(* CoDeSys 2.3.9.50 project: Acp_Bag_2Wrapping_Code.pro *)
(* Libraries: SysLibAlarmTrend.lib 17.10.05 13:12:38, TcBase.lib 14.5.09 12:14:08, TcSystem.lib 7.6.16 11:01:22, TcUtilities.lib 3.2.16 16:08:58, FB_DateTime.lib 15.2.16 16:36:26, STANDARD.LIB 5.6.98 12:03:02, TcEtherCAT.lib 30.11.16 19:52:18, COMlibV2.lib 24.2.14 12:45:46, SysLibTargetVisu.lib 16.6.08 16:24:26, TcBaseMath.lib 27.7.04 12:07:56, SysLibVisu.lib 7.7.04 18:17:22, TcSystemCX.lib 7.9.16 12:51:26, TcMath.lib 23.9.04 15:15:30 *)

(* Task configuration *)
TASK Standard (PRIORITY := 0, INTERVAL := T#10ms);
	MAIN
END_TASK

(* Global variable list: Alarms *)
VAR_GLOBAL
	bAError1: BOOL;
	bAError2: BOOL;
	bAError3: BOOL;
	bAError4: BOOL;
	bAError5: BOOL;
	bAError6: BOOL;
	bAError7: BOOL;
	bAError8: BOOL;
	bAError9: BOOL;
	bAError10: BOOL;
	bAError11: BOOL;
	bAError12: BOOL;
	bAError13: BOOL;
	bAError14: BOOL;
	bAError15: BOOL;
	bAError16: BOOL;
	bAError17: BOOL;
	bAError18: BOOL;
	bAError19: BOOL;
	bAError20: BOOL;
	bAError1Status: STRING;
	bAError2Status: STRING;
	bAError3Status: STRING;
	bAError4Status: STRING;
	bAError5Status: STRING;
	bAError6Status: STRING;
	bAError7Status: STRING;
	bAError8Status: STRING;
	bAError9Status: STRING;
	bAError10Status: STRING;
	bAError11Status: STRING;
	bAError12Status: STRING;
	bAError13Status: STRING;
	bAError14Status: STRING;
	bAError15Status: STRING;
	bAError16Status: STRING;
	bAError17Status: STRING;
	bAError18Status: STRING;
	bAError19Status: STRING;
	bAError20Status: STRING;
END_VAR

(* Global variable list: Auto *)
VAR_GLOBAL
	bQAFeedingConveyorMotor: BOOL;
	bAConeFeedConveyorStart: BOOL;
	bAConeFeedConWait: BOOL;
	bRConePresentInConeFeedCon: BOOL;

	bAConeFeedingPistonHomeRsError: BOOL;
	bQAConeFeedPisOn: BOOL;

	bASealConRdy: BOOL;
	bQAForwardPistonOn: BOOL;
	bQAReversePistonOn: BOOL;

	bAConeTiltingRdy: BOOL;
	ConeFeedPistonRdy: BOOL;
	bAConeFeedCount: BOOL;
	bAConeFeedPisOn: BOOL;
	bAConeFeedingPistonEndRsError: BOOL;
	Cone1Reached: BOOL;
	bAConeFeededCount: INT;
	Cone2Reached: BOOL;
	TotalNoOfCones: INT;

	bAConeFwdRevRdy: BOOL;
	bATiltingPistonOn: BOOL;
	bAConeTiltingPistonEndRsError: BOOL;
	bAFwdRevPisRdy: BOOL;
	bAFwdRevCom: BOOL;
	bAConeTiltingPistonHomeRsError: BOOL;
	bATiltingCylCom: BOOL;
	bAConeTiltingCount: INT;

	bAWrapRdy: BOOL;
	bAForwardPistonOn: BOOL;
	bAReversePistonOn: BOOL;
	bAForwardPisEndRsError: BOOL;
	bAReversePisEndRsError: BOOL;
	bAFwdRevCount: INT;
	bAForwardPisHomeRsError: BOOL;
	bAReversePisHomeRsError: BOOL;
	bAWrappingConRdy: BOOL;

	bAWrapConRdy: BOOL;
	bAWrappingConOn: BOOL;
	bAWrapConeAlaignError: BOOL;
	bAWrapConeAlaignError1: BOOL;
	bAWrappingPisRdy: BOOL;
	bAWrapPiston1On: BOOL;
	bAWrapPiston2On: BOOL;
	bASealingConRdy: BOOL;
	bASheetFeedError: BOOL;
	bAWrapPis1EndRsError: BOOL;
	bAWrapPis2EndRsError: BOOL;
	bAWrappingPisCylCom: BOOL;
	bAWrappingPisCylComInt: BOOL;
	bASealUnitStart: BOOL;


	iBagRowCounter_243: INT;
	bQAColumnStopperPiston: BOOL;
	bABagOperationStarted_243: BOOL;
	bABagUnitRdy_243: BOOL;
	bABagOperationRdy_243: BOOL;
	bQAConePusher2Piston: BOOL;
	bQAColumnReversePiston: BOOL;
	bQAConePusher1Piston: BOOL;
	bABagHalfOpCom_243: BOOL;
	bABagOperationStarted: BOOL;
	bABagOperationComplete: BOOL;
	bQABagHolder: BOOL;
	bQASeparatorplatePiston: BOOL;
	bQABagUp_Down50piston: BOOL;
	bABagOperationComplete_243: BOOL;
	bQABagPusherForwardPiston: BOOL;
	bQABagPusherReversePiston: BOOL;
	TON_bagPusher_243: TON;
	BagOpCom_243: BOOL;
	bForceBagHolder: BOOL;
	bABagComplete: BOOL;
	bQABagTiltingpistonReverse: BOOL;
	bABagTiltingRevOk_243: BOOL;
	bQAColumnConeReversePiston: BOOL;
	bQABagUp_Down180piston: BOOL;
	bQABagTiltingpistonForward: BOOL;
	bQABagBagUp_Down50piston: BOOL;
	bQABagRowHolderpiston: BOOL;

	bASealingConRdy_Bag: BOOL;
	bASealingConRdy_Box: BOOL;
	bASealingUnitOperationCom: BOOL;
	bABoxUnitRdy: BOOL;
	bABoxOperationCom: BOOL;
	bQASealingConFwd1: BOOL;
	bQASealingConRev: BOOL;
	bASealConeSet1Started: BOOL;
	bQASealingConFwd2: BOOL;
	bASealingConeCountEnable: BOOL;
	bASealConeSet1Completed: BOOL;
	bASealConeSet2Started: BOOL;
	bASealConeSet2Completed: BOOL;
	bASealConeRevSetCompleted: BOOL;
	bASealConeMissError: BOOL;
	bASealConeMissErrorStatus: STRING;
	bASealConeMissError1: BOOL;
	bASealConeMissError2: BOOL;
	bASealConeMissError3: BOOL;
	bASealingUnitInt: BOOL;
	bQASealingSeparatorYAxisPiston: BOOL;
	bQASealingTopPiston: BOOL;
	bQASealingBottomPiston: BOOL;
	bQASealingSeparatorXAxisPiston: BOOL;
END_VAR

(* Global variable list: DataLog *)
VAR_GLOBAL
	R_TRIG_IndoPrint: R_TRIG;
	FB_FileOpen_Indo: FB_FileOpen;
	FB_FileWrite_Indo: FB_FileWrite;
	FB_FileClose_Indo: FB_FileClose;
	FB_FileDelete_Indo: FB_FileDelete;
	IndoReport: INT;
	ReportHead1_Indo: BOOL;
	ST1_ProductionData: BOOL;
	ReportHead2_Indo: BOOL;
	ReportBot1_Indo: BOOL;
	stStation1_ProductionData: BOOL;
	ReportBot2_Indo: BOOL;
	testbit: BOOL;
	sOldDay: STRING;
	WriteError: INT;
	OpenError: INT;
	ProductionData_IndoPrint2:STRING(255);
	ProductionDataError_IndoPrint2:STRING(255);
	ProductionDataValues_IndoPrint_Com:STRING(255);
	bANewDay: BOOL;
	SerialNoError: DINT;
	ProductionDataValues_IndoPrint: STRING(255);
	ProductionData_IndoPrint: STRING(255);
	ProductionDataError_IndoPrint: STRING(255);
	ProductionData_ReportData1 : ProductionData_ReportData;
	PROCESSCOMPLETE: BOOL;
	ReportSave: BOOL;
	SerialNo AT %Q*: DINT;
END_VAR

(* Global variable list: Initialize *)
VAR_GLOBAL
	Initialize_TapHmi: BOOL;
	bAInitializeSeq: BOOL;
	bAMachineOn: BOOL;
	bASupplyPressureError: BOOL;
	IntAllOver: BOOL;
	bAIntHomeCheckError: BOOL;

	bQRWappingConveyorMotor: BOOL;
	WrappingConIntRunning: BOOL;
	WrapConIntOver: BOOL;
	bRConePresentInWrapCon: BOOL;
	bQRWrappingPiston1: BOOL;
	bQRWrappingPiston2: BOOL;
	bAWrappingPiston1RsError: BOOL;
	bAWrappingPiston2RsError: BOOL;
	WrapUnitIntOver: BOOL;
	sWrappingConStatus: STRING;
	TiltIntRdy: BOOL;

	bQRForwardPiston: BOOL;
	bQRReversePiston: BOOL;
	bQRTiltingPiston: BOOL;
	bQATiltingPiston: BOOL;
	TiltingIntOvr: BOOL;

	bQRSealingConveyorMotor: BOOL;
	bRConePresentInSealCon: BOOL;
	SealingConIntRunning: BOOL;
	sSealingConStatus: STRING;
	SealConIntOver: BOOL;
	bQRSealingTopPiston: BOOL;
	bQRSealingBottomPiston: BOOL;
	bQRSealingSeparatorXAxisPiston: BOOL;
	bRSealUnitIntOver: BOOL;
	bQRSealingSeparatorYAxisPiston: BOOL;

	bRBagUnitIntRdy: BOOL;
END_VAR

(* Global variable list: Inputs *)
VAR_GLOBAL
					(*I1-EL1809*)

	(*IR1*)	bIUnit_A_RowStopperHome AT %I* : BOOL;
	(*IR2*)	bIUnit_A_RowStopperMiddle AT %I* :BOOL;
	(*IR3*)	bIUnit_A_RowStopperEnd AT %I* :BOOL;
	(*IR4*)	bIUnit_B_RowStopperHome AT %I* :BOOL;
	(*IR5*)	bIUnit_B_RowStopperMiddle AT %I* :BOOL;
	(*IR6*)	bIUnit_B_RowStopperEnd AT %I* :BOOL;
	(*IR7*)	bIUnit_A_ConeDetectionSensor1 AT %I* :BOOL;
	(*IR8*)	bIUnit_A_ConeDetectionSensor2 AT %I* :BOOL;
	(*IR9*)	bIUnit_A_ConeDetectionSensor3 AT %I* :BOOL;
	(*IR10*)	bIUnit_A_ConeDetectionSensor4 AT %I* :BOOL;
	(*IR11*)	bIUnit_A_ConeCrossLimitSwitch AT %I* :BOOL;
	(*IR12*)	bIUnit_B_ConeDetectionSensor1 AT %I* :BOOL;
	(*IR13*)	bIUnit_B_ConeDetectionSensor2 AT %I* :BOOL;
	(*IR14*)	bIUnit_B_ConeDetectionSensor3 AT %I* :BOOL;
	(*IR15*)	bIUnit_B_ConeDetectionSensor4 AT %I* :BOOL;
	(*IR16*)	bIUnit_B_ConeCrossLimitSwitch AT %I* :BOOL;


					(*I2-EL1809*)

	(*IR17*)	bIUnit_AStartPb AT %I* :BOOL;
	(*IR18*)	bIUnit_BStartPb AT %I* :BOOL;
	(*IR19*)	bISpare1 AT %I* :BOOL;
	(*IW1*)	bIMcStartPb AT %I* :BOOL;
	(*IW2*)	bIMcStopPb AT %I* :BOOL;
	(*IW3*)	bIAutoManualSwitch AT %I* :BOOL;
	(*IW4*)	bIEmergencySwitchPb AT %I* :BOOL;
	(*IW5*)	bIProgramKeySwitch AT %I* :BOOL;
	(*IW6*)	bIConeOrientationTopLimitSwitch AT %I* :BOOL;
	(*IW7*)	bIFeedconeStopSensor AT %I* :BOOL;
	(*IW8*)	bIConeFeedingPistonHome AT%I* :BOOL;
	(*IW9*)	bIConeFeedingPistonEnd AT %I* :BOOL;
	(*IW10*)	bIForwardPistonHome AT %I* :BOOL;
	(*IW11*)	bIForwardPistonEnd AT %I* :BOOL;
	(*IW12*)	bIReversePistonHome AT %I* :BOOL;
	(*IW13*)	bIReversePistonEnd AT %I* :BOOL;

						(*I3-EL1809*)

	(*IW14*)	bITiltingHome AT %I* :BOOL;
	(*IW15*)	bITiltingMiddle AT %I* :BOOL;
	(*IW16*)	bITiltingEnd AT %I* :BOOL;
	(*IW17*)	bIWrappingChanelPiston1Home AT %I* :BOOL;
	(*IW18*)	bIWrappingChanelPiston1Middle AT %I* :BOOL;
	(*IW19*)	bIWrappingChanelPiston1End AT %I* :BOOL;
	(*IW20*)	bIWrappingChanelPiston2Home AT %I* :BOOL;
	(*IW21*)	bIWrappingChanelPiston2Middle AT %I* :BOOL;
	(*IW22*)	bIWrappingChanelPiston2End AT %I* :BOOL;
	(*IW23*)	bIWrappingCone1 AT %I* :BOOL;
	(*IW24*)	bIWrappingCone2 AT %I* :BOOL;
	(*IW25*)	bIFilmTensionRod1Home AT %I* :BOOL;
	(*IW26*)	bIFilmTensionRod1End AT %I* :BOOL;
	(*IW27*)	bIFilmTensionRod2Home AT %I* :BOOL;
	(*IW28*)	bIFilmTensionRod2End AT %I* :BOOL;
	(*IW29*)	bISpare2 AT %I* :BOOL;

						(*I4-EL1809*)

	(*IW30*)	bISealingSeparatorYAxisPistonHome AT %I* :BOOL;
	(*IW31*)	bISealingSeparatorYAxisPistoEnd AT %I* :BOOL;
	(*IW32*)	bISealingTopPistonHome AT %I* :BOOL;
	(*IW33*)	bISealingTopPistonEnd AT %I* :BOOL;
	(*IW34*)	bISealingBottomPistonHome AT %I* :BOOL;
	(*IW35*)	bISealingBottomPistonEnd AT %I* :BOOL;
	(*IW36*)	bISealingSeparatorXAxisPistonHome AT %I* :BOOL;
	(*IW37*)	bISealingSeparatorXAxisPistonEnd AT %I* :BOOL;
	(*IW38*)	bIManualSealingPb AT %I* :BOOL;
	(*IW39*)	bIConeCountsensor AT %I* :BOOL;
	(*IW40*)	bIPressureSwitch AT %I* :BOOL;
	(*IW41*)	bIResetPb AT %I* :BOOL;
	(*IW42*)	bIPausePb AT %I* :BOOL;
	(*IW43*)	bIConeCountSensorRev AT %I* :BOOL;
	(*IW44*)	bIConecountStopperPistonHome AT %I* :BOOL;
	(*IW45*)	bIConecountStopperPistonEnd AT%I* :BOOL;


						(*I5-EL1809*)

	(*IW46*)	bIResetSealingPb AT %I* :BOOL;
	(*IW47*)	bISpare4 AT %I* :BOOL;
	(*IW48*)	bISpare5 AT %I* :BOOL;
	(*IW49*)	bISpare6 AT %I* :BOOL;
	(*IW50*)	bISpare7 AT %I* :BOOL;
	(*IW51*)	bISpare8 AT %I* :BOOL;
	(*IW52*)	bISpare9 AT %I* :BOOL;
	(*IW53*)	bISpare10 AT %I*: BOOL;

					(*I6-EL1809*)

	(*IB1*)	bIColumnStopperPistonHome AT %I*: BOOL;
	(*IB2*)	bIColumnStopperPistonEnd AT %I*: BOOL;
	(*IB3*)	bIColumnReversePistonHome AT %I*: BOOL;
	(*IB4*)	bIColumnReversePistonEnd AT %I*: BOOL;
	(*IB5*)	bISeperatorPlatePistonHome AT %I*: BOOL;
	(*IB6*)	bISeperatorPlatePistonEnd AT %I*: BOOL;
	(*IB7*)	bIConePusher1PistonHome AT %I*: BOOL;
	(*IB8*)	bIConePusher1PistonEnd AT %I*: BOOL;
	(*IB9*)	bIConePusher1SaftyObjectSensor AT %I*: BOOL;
	(*IB10*)	bIBagUpDown180PistonHome AT %I*: BOOL;
	(*IB11*)	bIBagUpDown180PistonEnd AT %I*: BOOL;
	(*IB12*)	bIBagUpDown50PistonHome AT %I*: BOOL;
	(*IB13*)	bIBagUpDown50PistonEnd AT %I*: BOOL;
	(*IB14*)	bIBagPusherPistonHome AT %I*: BOOL;
	(*IB15*)	bIBagPusherPistonMiddle AT %I*: BOOL;
	(*IB16*)	bIBagPusherPistonEnd AT %I*: BOOL;

						(*I7-EL1809*)

	(*IB17*)	bIBagTiltingPistonHome AT %I*: BOOL;
	(*IB18*)	bIBagiltingPistonEnd AT %I*: BOOL;
	(*IB19*)	bIBagEmptyCheckObjectSensor AT %I*: BOOL;
	(*IB20*)	bIBagHolderOn  AT %I*: BOOL;
	(*IB21*)	bIBagResetPb AT %I*: BOOL;
	(*IB22*) 	bISpare11 AT %I*: BOOL;
	(*IB23*) 	bISpare12 AT %I*: BOOL;
	(*IB24*) 	bISpare13 AT %I*: BOOL;
END_VAR

(* Global variable list: Main *)
VAR_GLOBAL
	(****************START / STOP / PAUSE / RESUME***************)
	Start_TapHmi: BOOL;
	bAutoModeOn: BOOL;
	bMcStartInAuto: BOOL;
	bMcStopEnable: BOOL;
	Stop_TapHmi: BOOL;
	Pause_TapHmi: BOOL;
	bPauseSeq: BOOL;
	Resume_TapHmi: BOOL;
	Reset_TapHmi: BOOL;
	bErrorReset: BOOL;
	bMcStopEnable1: BOOL;
(*============== Auto/Manual Mode Selection Logic========================*)
	bManualModeOn: BOOL;
	bManualmode: BOOL;
	sMcStatus: STRING;
	bHidePopUp: BOOL;
	bManualModeOk_TapHmi: BOOL;
	bManualModeNOk_TapHmi: BOOL;
(*====================Logic for Model Selection===============*)
	BagSelect_TapHmi: BOOL;
	bAMainIntStarted: BOOL;
	bABoxModeSelected: BOOL;
	BoxSelect_TapHmi: BOOL;
	bABagModeSelected: BOOL;
	sPackingModeStatus: STRING;

	(****************DATE AND TIME***********)
	FB_DateTime_1: FB_DateTime;
	sHourPreFix: STRING;
	sHou: STRING;
	sDayPreFix: STRING;
	sDay: STRING;
	sMonthPreFix: STRING;
	sMonth: STRING;
	sDayF: STRING;
	sMonthF: STRING;
	sDayMonth: STRING;
	sDayF1: STRING;
	sMonthF1: STRING;
	sDayMonth1: STRING;
	sDayMonthYear: STRING;
	sDayMonthYear1: STRING;
	sDaateReport: STRING;
	ReportPath: STRING;
	ReportPath_Final: STRING;
	ReportPath_Final_1: STRING;
	ReportPath_Final_2: STRING;
	sDateReport: STRING;
	ReportPathError: STRING;
	ReportPath_FinalError: STRING;
	ReportPath_Final_1Error: STRING;
	ReportPath_Final_2Error: STRING;
	DateTimeVar: STRING;
	wTodayToHmiFinal: STRING;
(*===============Shift Calculation============*)
	bAShift1Hour: BOOL;
	bAShift2Hour: BOOL;
	bAShift3Hour: BOOL;
	Sfiht1From_Hmi  AT %Q*: WORD;
	Sfiht2From_Hmi  AT %Q*: WORD;
	Sfiht3From_Hmi  AT %Q*: WORD;
	Sfiht1To_Hmi AT %Q*: WORD;
	Sfiht2To_Hmi AT %Q*: WORD;
	Sfiht3To_Hmi AT %Q*: WORD;
	sShitStatus: STRING;
END_VAR

(* Global variable list: Manual *)
VAR_GLOBAL
	WrappingSafety: BOOL;
	SealingSafety: BOOL;
	bManualSealEnable: BOOL;
	bManualSealEnable2: BOOL;
	bMManualSealOn: BOOL;
	bQM_Cone_Sealing_Bottom_Piston: BOOL;
	bQM_Cone_Sealing_Top_Piston: BOOL;
	bHMI_Cone_Forward_Piston_On: BOOL;
	bQM_Cone_Forward_Piston: BOOL;
	bHMI_Cone_Feeding_Piston_On: BOOL;
	bQM_Cone_Feeding_Piston: BOOL;
	bHMI_Cone_Reverse_Piston_On: BOOL;
	bQM_Cone_Reverse_Piston: BOOL;
	bHMI_Cone_Tilting_Piston_On: BOOL;
	bQM_Cone_Tilting_Piston: BOOL;
	bQM_Cone_Tilting_Piston_Rev: BOOL;
	bHMI_Cone_Tilting_Piston_On_Rev: BOOL;
	bHMI_Cone_Wrapping_Piston_On: BOOL;
	bQM_Cone_Wrapping_Piston_Rev: BOOL;
	bQM_Cone_Wrapping_Piston_Fwd: BOOL;
	bHMI_Cone_Wrapping_Piston_On_Rev: BOOL;
	bHMI_Cone_Sealing_Top_Piston_On: BOOL;
	bHMI_Cone_Sealing_Bottom_Piston_On: BOOL;
	bHMI_Cone_Sealing_YAxis_Piston_On: BOOL;
	bQM_Cone_Sealing_YAxis_Piston: BOOL;
	bHMI_Cone_Sealing_XAxis_Piston_On: BOOL;
	bQM_Cone_Sealing_XAxis_Piston: BOOL;
	bHMI_Cone_Feeding_Conveyor_On: BOOL;
	bQM_Cone_Feeding_Conveyor: BOOL;
	bHMI_Cone_Wrapping_Conveyor_On: BOOL;
	bQM_Cone_Wrapping_Conveyor: BOOL;
	bHMI_Cone_Sealing_Conveyor_On: BOOL;
	bQM_Cone_Sealing_Conveyor: BOOL;
	bIConePusher1_On_Hmi: BOOL;
	bQMConePusher1: BOOL;
	bIConePusher2_On_Hmi: BOOL;
	bQMConePusher2: BOOL;
	bIConePusher3_On_Hmi: BOOL;
	bQMConePusher3: BOOL;
	bIBagPusherFwd_On_Hmi: BOOL;
	bQMBagPusherFwd: BOOL;
	bIBagPusherRev_On_Hmi: BOOL;
	bQMBagPusherRev: BOOL;
	bIUpDownPiston_1_On_Hmi: BOOL;
	bQMUpDownPiston_1: BOOL;
	bIUpDownPiston_2_On_Hmi: BOOL;
	bQMUpDownPiston_2: BOOL;
	bIBagTiltingFwd_On_Hmi: BOOL;
	bQMBagTiltingFwd: BOOL;
	bIBagTiltingRev_On_Hmi: BOOL;
	bQMBagTiltingRev: BOOL;
	bIColumn_Stopper_Piston_On_Hmi: BOOL;
	bQMColumnStopperPiston: BOOL;
	bIColumnConeForwardPiston_On_Hmi: BOOL;
	bQMColumnConeForwardPiston: BOOL;
	bIBagHolder_On: BOOL;
	bIBagHolder_On_Hmi: BOOL;
	bIBagPusherHome: BOOL;
	bQMBagHolderPiston: BOOL;
	bHMI_RetA_Fwd_On: BOOL;
	bHMI_RetA_Rev_On: BOOL;
	bQM_RetA_Rev: BOOL;
	bQM_RetA_Fwd: BOOL;
	bHMI_Ret_RevA_On: BOOL;

	bHMI_RetB_Fwd_On: BOOL;
	bHMI_RetB_Rev_On: BOOL;
	bQM_RetB_Rev: BOOL;
	bQM_RetB_Fwd: BOOL;
	bHMI_Ret_RevB_On: BOOL;
	bHMI_Cone_Wrapping_Piston1_On: BOOL;
	bQM_Cone_Wrapping_Piston1_Fwd: BOOL;
	bHMI_Cone_Wrapping_Piston1_On_Rev: BOOL;
	bQM_Cone_Wrapping_Piston1_Rev: BOOL;
	bHMI_Cone_Wrapping_Piston2_On: BOOL;
	bQM_Cone_Wrapping_Piston2_Rev: BOOL;
	bQM_Cone_Wrapping_Piston2_Fwd: BOOL;
	bHMI_Cone_Wrapping_Piston2_On_Rev: BOOL;
END_VAR

(* Global variable list: Outputs *)
VAR_GLOBAL
				(*O1-EL2809*)

	RetA_RowStopperMotorFwd AT %Q* :BOOL;(*OR1*)
	RetA_RowStopperMotorRev AT %Q* :BOOL;(*OR2*)
	RetB_RowStopperMotorFwd AT %Q* :BOOL;(*OR3*)
	RetB_RowStopperMotorRev AT %Q* :BOOL;(*OR4*)
	SpareOutput1 AT %Q* :BOOL;(*OR5*)
	RetA_WeightOk AT %Q* :BOOL;(*OR6*)
	RetA_WeightNOk AT %Q* :BOOL;(*OR7*)
	RetB_WeightOk AT %Q* :BOOL;(*OR8*)
	RetB_WeightNOk AT %Q* :BOOL;(*OR9*)
	SpareOutput2 AT %Q* :BOOL;(*OR10*)
	SpareOutput3 AT %Q* :BOOL;(*OR11*)
	SpareOutput4 AT %Q* :BOOL;(*OR12*)
	TowerLampRed AT %Q* :BOOL;(*R1*)
	TowerLampGreen AT %Q* :BOOL;(*R2*)
	TowerLampYellow AT %Q* :BOOL;(*R3*)
	TowerBuzzer AT %Q* :BOOL;(*R4*)


			(*O2-EL2809*)

	ConeFeedingPiston AT %Q* :BOOL;(*OW1*)
	ForwardPiston AT %Q* :BOOL;(*OW2*)
	ReversePiston AT %Q* :BOOL;(*OW3*)
	TiltingPiston AT %Q* :BOOL;(*OW4*)
	WrappingPiston1 AT %Q* :BOOL;(*OW5*)
	WrappingPiston2 AT %Q* :BOOL;(*OW6*)
	SealingSeparatorYAxisPiston AT %Q* :BOOL;(*OW7*)
	SealingTopPiston AT %Q* :BOOL;(*OW8*)
	SealingBottomPiston AT %Q* :BOOL;(*OW9*)
	SealingSeparatorXAxisPiston AT %Q* :BOOL;(*OW10*)
	FilmRollerMotor1 AT %Q* :BOOL;(*OW11*)
	FilmRollerMotor2 AT %Q* :BOOL;(*OW12*)
	ConeCountPiston AT %Q* :BOOL;(*OW13*)
	FeedingConveyorMotor AT %Q* :BOOL;(*OW14*)
	WappingConveyorMotor AT %Q* :BOOL;(*OW15*)
	SealingConveyorMotor AT %Q* :BOOL;(*OW16*)



			(*O3-EL2008*)

	SpareOutput5 AT %Q* :BOOL;(*OW20*)
	SpareOutput6 AT %Q* :BOOL;(*OW21*)
	SpareOutput7 AT %Q* :BOOL;(*OW22*)
	SpareOutput8 AT %Q* :BOOL;(*OW23*)
	SpareOutput9 AT %Q* :BOOL;(*OW24*)
	SpareOutput10 AT %Q* :BOOL;(*OW25*)
	SpareOutput11 AT %Q* :BOOL;(*OW26*)
	SpareOutput12 AT %Q* :BOOL;(*OW27*)

			(*O4-EL2809*)

	ColumnStopperPiston AT %Q* :BOOL;(*OB1*)
	ColumnReversePiston AT %Q* :BOOL;(*OB2*)
	SeparatorplatePiston AT %Q* :BOOL;(*OB3*)
	ConePusher1Piston AT %Q* :BOOL;(*OB4*)
	ConePusher2Piston AT %Q* :BOOL;(*OB5*)
	BagPusherForwardPiston AT %Q* :BOOL;(*OB6*)
	BagPusherReversePiston AT %Q* :BOOL;(*OB7*)
	BagHolderpiston AT %Q* :BOOL;(*OB8*)
	BagUp_Down180piston AT %Q* :BOOL;(*OB9*)
	BagUp_Down50piston AT %Q* :BOOL;(*OB10*)
	BagTiltingpistonForward AT %Q* :BOOL;(*OB11*)
	BagTiltingpistonReverse AT %Q* :BOOL;(*OB12*)
	BagRowHolderpiston AT %Q* :BOOL;(*OB13*)
	SpareOutput13 AT %Q* :BOOL;(*OB14*)
	SpareOutput14 AT %Q* :BOOL;(*OB15*)
	SpareOutput15 AT %Q* :BOOL;(*OB16*)

END_VAR

(* Global variable list: Parameters *)
VAR_GLOBAL
	Default_NetWeight_Report: STRING;
	Default_GrossWeight_Report: STRING;
	Actual_NetWeight_Report: STRING;
	Actual_GrossWeight_Report: STRING;
	COUNT_DIS: STRING;
	BLEND_DIS: STRING;
	LOTNO_DIS: STRING;
	CARTONNO_DIS: DINT;
	SHADE_DIS: STRING;
END_VAR

(* Global variable list: Print *)
VAR_GLOBAL
	PrintEnabled: BOOL;
	PrintValue: INT;
	PrintEnable_TogHmi: BOOL;
	ProductionData_PrintData: ProductionData_PrintData;
	ProductionDataValues_Print: STRING(255);
	ProductionDataValues_Print_Com:STRING(255);
	ProductionData_Print: STRING(255);
	FB_FileOpen1: FB_FileOpen;
	FB_FileWrite1: FB_FileWrite;
	FB_FileClose1: FB_FileClose;
	FB_FileDelete1: FB_FileDelete;
	PrintOk: BOOL;
END_VAR

(* Data type *)
TYPE ProductionData_PrintData :
STRUCT
	Print:STRING;
	ConeType1:STRING;
	Blend1:STRING;
	DefaultnetWt1:STRING;
	DefaultGrossWt1:STRING;
	LotNo1:STRING;
	BagNo1:STRING;
	Shade1:STRING;
END_STRUCT
END_TYPE

(* Data type *)
TYPE ProductionData_ReportData :
STRUCT
	SERIALNO			:STRING;
	SDATE				:STRING;
	STIME				:STRING;
	BAGNO				:STRING;
	COUNTCODE		:STRING;
	LOTNO				:STRING;
	DFLTNETWEIGHT	:STRING;
	ACTNETWEIGHT		:STRING;
	DFLTGROSSWEIGHT	:STRING;
	ACTGROSSWEIGHT	:STRING;
END_STRUCT
END_TYPE

(* POU MAIN, ST *)
PROGRAM MAIN
	VAR

END_VAR
					(*START / STOP / PAUSE / RESUME*)


	IF (bIMcStartPb OR Start_TapHmi)  AND bAutoModeOn  THEN
	 bMcStartInAuto:=TRUE;
	bMcStopEnable:=FALSE;
	END_IF

	IF  bIMcStopPb OR Stop_TapHmi  OR NOT bAutoModeOn OR NOT bIEmergencySwitchPb THEN
	 bMcStartInAuto:=FALSE;bMcStopEnable:=TRUE;bMcStopEnable1:=TRUE;
	ELSE bMcStopEnable1:=TRUE;
	 END_IF

	IF Pause_TapHmi THEN
	bPauseSeq:=TRUE;END_IF
	IF Resume_TapHmi THEN
	bPauseSeq:=FALSE;END_IF

	IF bIResetPb OR Reset_TapHmi  OR bIResetSealingPb THEN
	bErrorReset:=TRUE;
	ELSE bErrorReset:=FALSE;END_IF

					(*============== Auto/Manual Mode Selection Logic========================*)

		IF bIAutoManualSwitch THEN
			bAutoModeOn:=TRUE; bManualModeOn:=FALSE;
		ELSIF  bManualmode  THEN
			bManualModeOn:=TRUE; bAutoModeOn:=FALSE;
		END_IF

		IF bManualModeOn THEN sMcStatus:='Machine in Manual Mode';
		ELSIF bAutoModeOn THEN sMcStatus:='Machine in Auto Mode';
		END_IF

	IF bMcStartInAuto  AND NOT  bIAutoManualSwitch THEN
	bHidePopUp:=TRUE; END_IF

	IF NOT  bMcStartInAuto  AND NOT  bIAutoManualSwitch THEN
	bManualmode:=TRUE;  END_IF

	IF bHidePopUp AND bManualModeOk_TapHmi THEN
	bManualmode:=TRUE;bAutoModeOn:=FALSE;bHidePopUp:=FALSE; END_IF

	IF bHidePopUp AND bManualModeNOk_TapHmi THEN
	bHidePopUp:=FALSE; END_IF

					 (*====================Logic for Model Selection===============*)

		IF bAutoModeOn AND BagSelect_TapHmi AND NOT bAMainIntStarted THEN
		bABoxModeSelected:=FALSE;BoxSelect_TapHmi:=FALSE;bABagModeSelected:=TRUE; BoxSelect_TapHmi:=FALSE;
		ELSIF bAutoModeOn AND   BoxSelect_TapHmi AND NOT bAMainIntStarted THEN
		bABagModeSelected:=FALSE; BagSelect_TapHmi:=FALSE;bABoxModeSelected:=TRUE;
		END_IF

		IF bABagModeSelected THEN sPackingModeStatus:=' Bag Packing Selected '; END_IF
		IF bABoxModeSelected THEN sPackingModeStatus:=' Carton Packing Selected  '; END_IF




			(****************DATE AND TIME***********)

(*======================= RTC==============================*)

FB_DateTime_1(NET_ID:='5.62.177.154.1.1 ' , DATE_TIME=> );

IF FB_DateTime_1.FBLTIME.systemTime.wHour >0 AND  FB_DateTime_1.FBLTIME.systemTime.wHour<9 THEN
sHourPreFix:='0';sHou:=CONCAT(STR1:=sHourPreFix, Str2:=WORD_TO_STRING(FB_DateTime_1.FBLTIME.systemTime.wHour));
ELSIF FB_DateTime_1.FBLTIME.systemTime.wHour >=10 AND  FB_DateTime_1.FBLTIME.systemTime.wHour<=24 THEN
sHou:=WORD_TO_STRING(FB_DateTime_1.FBLTIME.systemTime.wHour);
END_IF

IF FB_DateTime_1.FBLTIME.systemTime.wDay >0 AND  FB_DateTime_1.FBLTIME.systemTime.wDay<10 THEN
sDayPreFix:='0';sDay:=CONCAT(STR1:=sDayPreFix, Str2:=WORD_TO_STRING(FB_DateTime_1.FBLTIME.systemTime.wDay));
ELSIF FB_DateTime_1.FBLTIME.systemTime.wDay >=10 AND  FB_DateTime_1.FBLTIME.systemTime.wDay<=31 THEN
sDay:=WORD_TO_STRING(FB_DateTime_1.FBLTIME.systemTime.wDay);
END_IF

IF FB_DateTime_1.FBLTIME.systemTime.wMonth >0 AND  FB_DateTime_1.FBLTIME.systemTime.wMonth<10 THEN
sMonthPreFix:='0';sMonth:=CONCAT(STR1:=sMonthPreFix, Str2:=WORD_TO_STRING(FB_DateTime_1.FBLTIME.systemTime.wMonth));
ELSIF FB_DateTime_1.FBLTIME.systemTime.wMonth >=10 AND  FB_DateTime_1.FBLTIME.systemTime.wMonth<=12 THEN
sMonth:=WORD_TO_STRING(FB_DateTime_1.FBLTIME.systemTime.wMonth);
END_IF

sDayF1:=CONCAT(STR1:=sDay, STR2:=':');
sMonthF1:=CONCAT(STR1:=sMonth, STR2:=':');
sDayMonth1:=CONCAT(STR1:=sDayF1, STR2:=sMonthF1);
sDayMonthYear1:=CONCAT(STR1:=sDayMonth1, STR2:=WORD_TO_STRING(FB_DateTime_1.FBLTIME.systemTime.wYear));

sDaateReport:=(sDayMonthYear1);

sDayF:=CONCAT(STR1:=sDay, STR2:='_');
sMonthF:=CONCAT(STR1:=sMonth, STR2:='_');
sDayMonth:=CONCAT(STR1:=sDayF, STR2:=sMonthF);
sDayMonthYear:=CONCAT(STR1:=sDayMonth, STR2:=WORD_TO_STRING(FB_DateTime_1.FBLTIME.systemTime.wYear));

ReportPath:=CONCAT(STR1:='ProductionData', STR2:='_');
ReportPath_Final:=CONCAT(STR1:=ReportPath, STR2:=sDayMonthYear);

ReportPath_Final_1:=CONCAT(STR1:='\\computer-PC\Reports\', STR2:=ReportPath_Final);
ReportPath_Final_2:=CONCAT(STR1:=ReportPath_Final_1, STR2:='.csv');

sDayF1:=CONCAT(STR1:=sDay, STR2:=':');
sMonthF1:=CONCAT(STR1:=sMonth, STR2:=':');
sDayMonth1:=CONCAT(STR1:=sDayF1, STR2:=sMonthF1);
sDayMonthYear1:=CONCAT(STR1:=sDayMonth1, STR2:=WORD_TO_STRING(FB_DateTime_1.FBLTIME.systemTime.wYear));

sDateReport:=(sDayMonthYear1);

sDayF:=CONCAT(STR1:=sDay, STR2:='_');
sMonthF:=CONCAT(STR1:=sMonth, STR2:='_');
sDayMonth:=CONCAT(STR1:=sDayF, STR2:=sMonthF);
sDayMonthYear:=CONCAT(STR1:=sDayMonth, STR2:=WORD_TO_STRING(FB_DateTime_1.FBLTIME.systemTime.wYear));

ReportPathError:=CONCAT(STR1:='ErrorData', STR2:='_');
ReportPath_FinalError:=CONCAT(STR1:=ReportPathError, STR2:=sDayMonthYear);

ReportPath_Final_1Error:=CONCAT(STR1:='\\computer-PC\Reports\', STR2:=ReportPath_FinalError);
ReportPath_Final_2Error:=CONCAT(STR1:=ReportPath_Final_1Error, STR2:='.csv');

DateTimeVar:=FB_DateTime_1.DATE_TIME;



					(*===============Shift Calculation============*)


IF FB_DateTime_1.FBLTIME.systemTime.wHour >= Sfiht1From_Hmi AND FB_DateTime_1.FBLTIME.systemTime.wHour<=Sfiht1To_Hmi THEN
bAShift1Hour:=TRUE;
ELSE
bAShift1Hour:=FALSE;
END_IF



IF FB_DateTime_1.FBLTIME.systemTime.wHour>=Sfiht2From_Hmi AND FB_DateTime_1.FBLTIME.systemTime.wHour <= Sfiht2To_Hmi THEN

bAShift2Hour:=TRUE;
ELSE
bAShift2Hour:=FALSE;
END_IF


IF FB_DateTime_1.FBLTIME.systemTime.wHour>=  Sfiht3From_Hmi AND FB_DateTime_1.FBLTIME.systemTime.wHour<=  Sfiht3To_Hmi THEN

bAShift3Hour:=TRUE;
ELSE
bAShift3Hour:=FALSE;
END_IF

IF bAShift1Hour THEN sShitStatus:='SHIFT - 1';
ELSIF bAShift2Hour THEN sShitStatus:='SHIFT - 2';
ELSIF bAShift3Hour THEN sShitStatus:='SHIFT - 3';
END_IF

Bag_Unit();
ConeFeedCon();
ConeFeedPiston();
Forward_Reverse_Piston();
Ret_A();
Ret_B();
Sealing_Unit();
Tilting_Piston();
Wrapping_Unit();
ErrorData_Report();
Print_Report();
ProductionData_Report();
Bag_Int();
ConeFeedCon_Int();
ConeTransfer_Int();
Main_Int();
Ret_Int();
Sealing_Int();
Wrapping_Int();
Manual();
Weight_Read();
END_PROGRAM

(* POU Auto/Bag_Unit, ST *)
PROGRAM Bag_Unit
VAR
	step: INT;
	iBagRowCounter_243: INT;
	TON_ConeFeedFwdOffDly_1_243: TON;
	TON_Count_243: TON;
	TON_ConePusherOffDly_243: TON;
	TON_ConeFeedFwdOffDly_243: TON;
	TON_ConePusherOnDly_243: TON;
	TON_ConePusherOffDly_2_243: TON;
	TON_ConeFeedFwdOffDly_3_243: TON;
	TON_ConePusherOnDly_2_243: TON;
	TON_ConePusherOnDly_3_243: TON;
	TON_bagPusher_243: TON;
	BagTilting_Blink2_243: TON;
	BagTilting_Blink1_243: TON;

END_VAR
CASE step OF

0:IF IntAllOver AND bABagModeSelected THEN iBagRowCounter_243:= 0; step:=step+1;END_IF

1:	iBagRowCounter_243:= 0; step:=step+1;

2:	bQAColumnConeReversePiston:=FALSE;
	IF bIColumnReversePistonHome AND NOT bPauseSeq THEN
	TON_ConeFeedFwdOffDly_1_243(IN:=FALSE); step := step +1;END_IF

3:	TON_ConeFeedFwdOffDly_1_243(IN:=TRUE , PT:=t#0.1s , Q=> , ET=> );
	IF  TON_ConeFeedFwdOffDly_1_243.Q THEN step := step +1;END_IF

4:	TON_ConeFeedFwdOffDly_1_243(IN:=FALSE);bQAColumnStopperPiston:=TRUE;
	IF  bIColumnStopperPistonEnd AND NOT bPauseSeq THEN
		 bABagOperationStarted_243:= FALSE;bABagUnitRdy_243:=TRUE;
		step := step +1;
	END_IF

5:	IF bABagOperationRdy_243  AND NOT bPauseSeq THEN
	 iBagRowCounter_243:=iBagRowCounter_243+1;bABagOperationStarted_243:=TRUE;
	bABagOperationRdy_243:=FALSE; step:=step+1;
	END_IF

6:	TON_Count_243(IN:=FALSE);bABagOperationRdy_243:=FALSE;
	IF (iBagRowCounter_243 = 1 OR iBagRowCounter_243= 2 OR iBagRowCounter_243 = 3 OR iBagRowCounter_243 = 4 ) AND NOT bPauseSeq THEN
	step:=step+1;

	ELSIF  ( iBagRowCounter_243 = 5 OR  iBagRowCounter_243 = 6 OR  iBagRowCounter_243 = 7 OR iBagRowCounter_243 = 8 ) AND NOT bPauseSeq THEN
	step := 19;
	END_IF

7:	IF   bISeperatorPlatePistonHome AND bIConePusher1PistonHome AND bIBagPusherPistonHome AND bIBagUpDown50PistonEnd
	AND bIBagUpDown180PistonEnd AND bIColumnStopperPistonEnd AND NOT bQABagHolder  AND NOT bPauseSeq THEN
	bQAConePusher2Piston:=FALSE;
	step := step +1;
	END_IF

8:	TON_ConePusherOffDly_243(IN:=TRUE , PT:=t#1s , Q=> , ET=> );
	IF TON_ConePusherOffDly_243.Q  AND NOT bPauseSeq  THEN
	bQAColumnReversePiston:=TRUE;
	TON_ConeFeedFwdOffDly_243(IN:=TRUE , PT:=t#0.1s , Q=> , ET=> );
	IF  TON_ConeFeedFwdOffDly_243.Q AND  bIColumnReversePistonEnd THEN step := step +1;END_IF
	END_IF

9:	TON_ConePusherOffDly_243(IN:=FALSE);
	IF  NOT bPauseSeq  THEN bQAColumnStopperPiston:=FALSE;step := step +1;END_IF

10:	TON_ConeFeedFwdOffDly_243(IN:=FALSE);
	IF bIColumnStopperPistonHome AND NOT bPauseSeq  THEN TON_ConePusherOnDly_243(IN:=TRUE , PT:=t#0.2s , Q=> , ET=> );
	IF TON_ConePusherOnDly_243.Q AND NOT bPauseSeq THEN
 		bQAConePusher1Piston:= TRUE ;bQAColumnReversePiston:=FALSE;step := step +1;
	END_IF END_IF

11: TON_ConePusherOnDly_243(IN:=FALSE);
	 IF bIConePusher1PistonEnd AND bIColumnReversePistonHome AND NOT bPauseSeq THEN
		bQAConePusher2Piston:= TRUE;bABagHalfOpCom_243:=TRUE;step := step +1;
	END_IF

12:	TON_ConePusherOnDly_243(IN:=TRUE , PT:=t#1.5s , Q=> , ET=> );
	IF TON_ConePusherOnDly_243.Q  AND NOT bPauseSeq  THEN bQAConePusher1Piston:= FALSE;
			step := step +1;
	END_IF

13:	TON_ConePusherOnDly_243(IN:=FALSE);
	 IF bIConePusher1PistonHome AND  (iBagRowCounter_243 = 1 OR iBagRowCounter_243 = 2  OR  iBagRowCounter_243 = 3 )
	AND NOT bQABagHolder  AND NOT bPauseSeq THEN
	bQAColumnStopperPiston:=TRUE;
		IF bIColumnStopperPistonEnd AND NOT bPauseSeq THEN
		 bABagOperationStarted:= FALSE;bABagOperationComplete:=TRUE;
		step := 2;END_IF

		ELSIF bIConePusher1PistonHome AND iBagRowCounter_243 =4  AND NOT bQABagHolder  AND NOT bPauseSeq THEN bQAColumnStopperPiston:=FALSE;
		IF  bIColumnStopperPistonHome AND NOT bPauseSeq THEN
		bABagOperationStarted_243:= FALSE;bABagOperationComplete_243:=TRUE;
		step :=14 ;END_IF
	END_IF

14:	step := step +1;

15:	IF   bISeperatorPlatePistonHome AND  bIConePusher1PistonHome AND bIBagPusherPistonHome AND NOT bPauseSeq AND NOT bQABagHolder THEN
	bQABagUp_Down180piston:=FALSE; step := step+1;bQAColumnStopperPiston:=TRUE;

	END_IF

16:	 IF bIBagUpDown180PistonHome AND bISeperatorPlatePistonHome AND bIConePusher1PistonHome AND NOT bQABagHolder  AND NOT bPauseSeq THEN
	bQASeparatorplatePiston:= TRUE ;bQABagUp_Down50piston:=FALSE;step := step +1;
	END_IF

17:	 IF bISeperatorPlatePistonEnd AND bIConePusher1PistonHome AND bIBagPusherPistonHome AND bIBagUpDown180PistonHome
	AND bIColumnStopperPistonEnd AND NOT bQABagHolder  AND NOT bPauseSeq THEN
	bQABagTiltingpistonForward:=TRUE;bQABagBagUp_Down50piston:=TRUE;bQABagTiltingpistonReverse:=FALSE;
	step := step +1;END_IF

18:	bQAColumnStopperPiston:=TRUE;
	 IF bISeperatorPlatePistonEnd AND bIConePusher1PistonHome AND bIBagPusherPistonHome AND bIBagUpDown50PistonEnd AND bIColumnStopperPistonEnd
	AND NOT bQABagHolder  AND NOT bPauseSeq THEN
	step := 2;END_IF

19:	bQAConePusher2Piston:= FALSE;step := step +1;


20:	TON_ConePusherOffDly_2_243(IN:=TRUE , PT:=t#1s , Q=> , ET=> );
	IF TON_ConePusherOffDly_2_243.Q  AND NOT bPauseSeq  THEN step := step +1;
	END_IF

21:	TON_ConePusherOffDly_2_243(IN:=FALSE);
	 IF bISeperatorPlatePistonEnd AND bIConePusher1PistonHome AND bIBagPusherPistonHome AND
	bIBagUpDown50PistonEnd AND bIColumnStopperPistonEnd AND
	bIColumnReversePistonHome AND NOT bQABagHolder  AND NOT bPauseSeq THEN
	bQAColumnReversePiston:=TRUE;step := step +1;END_IF

22:	TON_ConeFeedFwdOffDly_3_243(IN:=TRUE , PT:=t#0.1s , Q=> , ET=> );
	IF  TON_ConeFeedFwdOffDly_3_243.Q AND  bIColumnReversePistonEnd THEN step := step +1;END_IF

23:	TON_ConeFeedFwdOffDly_3_243(IN:=FALSE);bQAColumnStopperPiston:=FALSE;step := step +1;

24:	IF bIColumnStopperPistonHome AND NOT bPauseSeq  THEN TON_ConePusherOnDly_2_243(IN:=TRUE , PT:=t#0.2s , Q=> , ET=> );
	IF TON_ConePusherOnDly_2_243.Q AND NOT bPauseSeq THEN
	bQAConePusher1Piston:= TRUE ;bQAColumnReversePiston:=FALSE;step := step +1;
	END_IF END_IF
25:	TON_ConePusherOnDly_2_243(IN:=FALSE);
	 IF bIConePusher1PistonEnd AND bIColumnReversePistonHome AND NOT bQABagHolder  AND NOT bPauseSeq THEN
	bQAConePusher2Piston:= TRUE;bABagHalfOpCom_243:=TRUE;step := step +1;
	END_IF

26:	TON_ConePusherOnDly_3_243(IN:=TRUE , PT:=t#1.5s , Q=> , ET=> );
	IF TON_ConePusherOnDly_3_243.Q  AND NOT bPauseSeq  THEN
			step := step +1;
	END_IF

27:TON_ConePusherOnDly_3_243(IN:=FALSE);
	 IF bIConePusher1PistonEnd AND (iBagRowCounter_243 = 5 OR iBagRowCounter_243 = 6 OR iBagRowCounter_243 = 7  )
	AND NOT bQABagHolder  AND NOT bPauseSeq THEN
	bQAConePusher1Piston:= FALSE;step := step +1;
	ELSIF
	 bIConePusher1PistonEnd AND iBagRowCounter_243 = 8  AND NOT bQABagHolder  AND NOT bPauseSeq THEN
	step := 29;
	END_IF

28:IF  bIConePusher1PistonHome AND bIColumnStopperPistonHome THEN  bQAColumnStopperPiston:=TRUE;
	bABagOperationStarted_243:= FALSE; bABagOperationComplete_243:=TRUE;
	step := 2;END_IF

29: IF bIConePusher1PistonEnd AND bIBagUpDown50PistonEnd   AND NOT  bQABagHolder AND NOT bPauseSeq THEN
	bQABagPusherForwardPiston:=TRUE;bQABagPusherReversePiston:=FALSE;step := step +1;END_IF

30:TON_bagPusher_243(IN:=TRUE , PT:=t#0.4s , Q=> , ET=> );
	IF (TON_bagPusher_243.Q OR bIBagPusherPistonMiddle) THEN bQABagPusherForwardPiston:=FALSE;bQABagPusherReversePiston:=FALSE; step := step +1;END_IF

31:	TON_bagPusher_243(IN:=FALSE);
	bQABagPusherForwardPiston:=FALSE;bQABagPusherReversePiston:=FALSE;step := step +1;(*END_IF*)

32:	IF NOT bQABagHolder AND NOT bPauseSeq THEN bQASeparatorplatePiston:= FALSE;step := step +1;END_IF

33:	 IF   bISeperatorPlatePistonHome AND NOT bQABagHolder AND NOT bPauseSeq THEN
	 bQAConePusher1Piston:= FALSE;BagOpCom_243:=TRUE;step := step +1;END_IF

34:	IF   bIConePusher1PistonHome AND NOT bPauseSeq THEN
	bQAColumnStopperPiston:=TRUE;
	IF  bIColumnStopperPistonEnd THEN bABagOperationStarted_243:= FALSE;
	bABagOperationComplete_243:=TRUE;bQABagPusherReversePiston:=TRUE;step := step +1;END_IF
	END_IF

35:  IF   bISeperatorPlatePistonHome AND bIConePusher1PistonHome AND bIBagPusherPistonHome AND NOT bPauseSeq AND bIBagiltingPistonEnd THEN
	bQABagUp_Down50piston:=FALSE;step := step +1;END_IF

36:	 IF   bISeperatorPlatePistonHome AND bIConePusher1PistonHome AND bIBagPusherPistonHome AND NOT bPauseSeq AND  bIBagiltingPistonEnd AND
	bIBagUpDown180PistonHome AND bIBagUpDown50PistonHome THEN
	bQABagPusherForwardPiston:=TRUE;bQABagPusherReversePiston:=FALSE;
	IF NOT bIBagPusherPistonMiddle OR bErrorReset THEN bForceBagHolder:=TRUE;step := step +1;END_IF
	END_IF

37:	IF bIBagPusherPistonEnd AND  NOT bPauseSeq THEN
	bQABagPusherForwardPiston:=FALSE;bForceBagHolder:=FALSE;
	bQABagPusherReversePiston:=TRUE;step := step +1;END_IF

38:	IF bIBagPusherPistonHome AND  NOT bPauseSeq THEN
	bQABagPusherForwardPiston:=FALSE;bQABagPusherReversePiston:=FALSE;
	bQABagTiltingpistonForward:=FALSE;bABagTiltingRevOk_243:=TRUE;
	bQABagTiltingpistonReverse:=FALSE;
	step := step +1;END_IF

39: 	IF BagTilting_Blink1_243.Q  AND NOT bPauseSeq THEN
	bQABagTiltingpistonForward:=FALSE; bQABagTiltingpistonReverse:=TRUE;
	ELSE bQABagTiltingpistonReverse:=FALSE;
	IF bIBagTiltingPistonHome THEN bQABagTiltingpistonReverse:=FALSE;bABagTiltingRevOk_243:=FALSE;
	BagTilting_Blink1_243(IN:=FALSE);BagTilting_Blink2_243(IN:=FALSE);step:= step +1;END_IF END_IF


40:	IF bIBagTiltingPistonHome AND  NOT bPauseSeq THEN bQABagTiltingpistonForward:=FALSE;bQABagTiltingpistonReverse:=FALSE;
	bQABagUp_Down180piston:=TRUE;bQABagUp_Down50piston:=TRUE;
	step := step +1;END_IF

41:	IF bIBagResetPb THEN bABagComplete:= TRUE;step:=0;END_IF

END_CASE


IF (bIBagHolder_On OR bIBagHolder_On_Hmi ) AND bISeperatorPlatePistonHome AND bIConePusher1PistonHome THEN

bQABagHolder:=TRUE;ELSE bQABagHolder:=FALSE;END_IF

bQABagRowHolderpiston:=bQABagHolder;

BagTilting_Blink1_243(IN:=(bABagTiltingRevOk_243 AND NOT bIBagTiltingPistonHome AND NOT BagTilting_Blink1_243.Q)   , PT:=t#0.6s , Q=> , ET=> );
BagTilting_Blink2_243(IN:=BagTilting_Blink1_243.Q , PT:=t#0.9s , Q=> , ET=> );

IF bIBagTiltingPistonHome THEN bQABagTiltingpistonReverse := FALSE;END_IF
END_PROGRAM

(* POU Auto/ConeFeedCon, ST *)
PROGRAM ConeFeedCon
VAR

END_VAR
bQAFeedingConveyorMotor:=bAConeFeedConveyorStart;

IF bMcStopEnable AND NOT bRConePresentInConeFeedCon AND NOT bAConeFeedConWait AND NOT bPauseSeq THEN
	bAConeFeedConveyorStart:=TRUE;
ELSE bAConeFeedConveyorStart:=FALSE;END_IF




IF 	((IntAllOver AND bIFeedconeStopSensor AND NOT bIConeFeedingPistonHome) OR
	(IntAllOver AND bIFeedconeStopSensor AND bIConeOrientationTopLimitSwitch))  THEN
	bAConeFeedConWait:=TRUE;
	ELSE bAConeFeedConWait:=FALSE;END_IF

IF bMcStopEnable1 OR NOT bAutoModeOn  THEN
bAConeFeedConveyorStart:=FALSE;
bAConeFeedConWait:=FALSE;
bRConePresentInConeFeedCon:=FALSE;
END_IF
END_PROGRAM

(* POU Auto/ConeFeedPiston, ST *)
PROGRAM ConeFeedPiston
VAR
	ConeFeedPis: INT;
	ConeFeedCount: INT;
	R_TRIG_1: R_TRIG;
	TON_1: TON;
	ConeFeedCounter: CTU;

END_VAR
IF IntAllOver  AND bIConeOrientationTopLimitSwitch AND bIConeFeedingPistonHome AND NOT bPauseSeq   THEN
ConeFeedPistonRdy:=TRUE;
ELSE
ConeFeedPistonRdy:=FALSE;
END_IF

CASE ConeFeedCount OF

0:	R_TRIG_1(CLK:=ConeFeedPistonRdy , Q=> );
		IF R_TRIG_1.Q THEN TON_1(IN:= FALSE); ConeFeedCount:=ConeFeedCount+1; END_IF

1:	IF NOT bPauseSeq  THEN   bAConeFeedCount :=TRUE;
		 ConeFeedCount:=ConeFeedCount+1;END_IF

2:	TON_1(IN :=  TRUE  , PT:=t#1s , Q=> , ET=> );
		IF TON_1.Q THEN  ConeFeedCount:=ConeFeedCount+1; END_IF

3:	bAConeFeedCount :=FALSE;ConeFeedCount:=ConeFeedCount+1;

4: 	IF bIConeFeedingPistonEnd THEN
		ConeFeedCount:=ConeFeedCount+1; END_IF

5:	IF bIConeFeedingPistonHome THEN  ConeFeedCount:=0; END_IF

END_CASE


ConeFeedCounter(
	CU:=bAConeFeedCount  ,
	RESET:=bMcStopEnable  ,
	PV:=TotalNoOfCones,
	Q=> ,
	CV=> );


bQAConeFeedPisOn:=bAConeFeedPisOn;

CASE ConeFeedPis OF

0:	 IF IntAllOver  AND NOT bPauseSeq AND bAConeTiltingRdy THEN
	ConeFeedCounter.RESET:=FALSE;ConeFeedPis:=ConeFeedPis+1;END_IF

1:	IF bATiltingCylCom AND NOT bPauseSeq  THEN
	ConeFeedPis:=ConeFeedPis+1;END_IF

2:	IF ConeFeedCounter.CV=1 AND bIConeFeedingPistonHome  AND NOT bAConeFeedingPistonHomeRsError
	AND NOT bPauseSeq AND bITiltingHome THEN
	bAConeFeedPisOn:=TRUE;bATiltingCylCom:=FALSE;ConeFeedPis:=ConeFeedPis+1;END_IF

3:	IF  bIConeFeedingPistonEnd  AND  NOT bAConeFeedingPistonEndRsError AND NOT bPauseSeq THEN
		bAConeFeedPisOn:=FALSE;
		Cone1Reached:=TRUE;
		bAConeFeededCount:=bAConeFeededCount+1;
		ConeFeedPis:=ConeFeedPis+1;END_IF

4:	IF ConeFeedCounter.CV=2 AND bIConeFeedingPistonHome AND NOT bAConeFeedingPistonHomeRsError
	AND NOT bPauseSeq AND (bITiltingMiddle OR bITiltingEnd) THEN
	bAConeFeedPisOn:=TRUE;ConeFeedPis:=ConeFeedPis+1;END_IF

5:	IF  bIConeFeedingPistonEnd  AND  NOT bAConeFeedingPistonEndRsError AND NOT bPauseSeq THEN
		bAConeFeedPisOn:=FALSE;
		Cone2Reached:=TRUE;
		bAConeFeededCount:=bAConeFeededCount+1;
		ConeFeedCounter.RESET:=TRUE;
		ConeFeedPis:=ConeFeedPis+1;END_IF

6:	IF bAConeFeededCount = TotalNoOfCones THEN bAConeFeededCount:=bAConeFeededCount+1;
	ELSIF bAConeFeededCount < TotalNoOfCones THEN bAConeFeededCount:=bAConeFeededCount+2;END_IF

7:	bAConeFeededCount:=0;ConeFeedPis:=ConeFeedPis+1;

8:	ConeFeedCounter.RESET:=FALSE;ConeFeedPis:=1;

END_CASE




IF bMcStopEnable1 OR NOT bAutoModeOn  THEN
ConeFeedPistonRdy:=FALSE;
ConeFeedCount:=0;bAConeFeedCount :=FALSE;
ConeFeedPis:=0;bAConeFeededCount:=0;END_IF
END_PROGRAM

(* POU Auto/Forward_Reverse_Piston, ST *)
PROGRAM Forward_Reverse_Piston
VAR
	FwdRevPis: INT;


END_VAR
bQAForwardPistonOn:=bAForwardPistonOn;
bQAReversePistonOn:=bAReversePistonOn;
CASE FwdRevPis OF

0: IF IntAllOver  AND NOT bPauseSeq AND bAWrapRdy THEN
	FwdRevPis:=FwdRevPis+1;END_IF

1:	FwdRevPis:=FwdRevPis+1;

2:	IF bAFwdRevPisRdy AND (bASealConRdy OR bAWrapRdy) AND NOT bPauseSeq THEN
	bAForwardPistonOn:=TRUE;bAReversePistonOn:=TRUE;bASealConRdy:=FALSE;bAWrapRdy:=FALSE;
	bAFwdRevPisRdy:=FALSE;FwdRevPis:=FwdRevPis+1;END_IF

3:	IF bIForwardPistonEnd AND bIReversePistonEnd AND NOT bAForwardPisEndRsError
	AND NOT bAReversePisEndRsError AND NOT bPauseSeq THEN
	bAFwdRevCount:=bAFwdRevCount+2;
	bAForwardPistonOn:=FALSE;bAReversePistonOn:=FALSE;bAWrappingConRdy:=TRUE;
	FwdRevPis:=FwdRevPis+1;END_IF

4:	IF bIForwardPistonHome AND bIReversePistonHome AND NOT bPauseSeq
	AND NOT bAForwardPisHomeRsError AND NOT bAReversePisHomeRsError THEN
	bAFwdRevCom:=TRUE;FwdRevPis:=FwdRevPis+1;END_IF

5:	IF bAFwdRevCount >= TotalNoOfCones THEN bAFwdRevCount:=0;FwdRevPis:=FwdRevPis+1;
	ELSE FwdRevPis:=FwdRevPis+1;END_IF

6: 	FwdRevPis:=1;

END_CASE


IF bMcStopEnable1 OR NOT bAutoModeOn  THEN
FwdRevPis:=0;bAFwdRevCount:=0;bAFwdRevCom:=FALSE;
bAForwardPistonOn:=FALSE;bAReversePistonOn:=FALSE;
bAFwdRevPisRdy:=FALSE;IntAllOver:=FALSE;END_IF
END_PROGRAM

(* POU Auto/Ret_A, ST *)
PROGRAM Ret_A
VAR
END_VAR
;
END_PROGRAM

(* POU Auto/Ret_B, ST *)
PROGRAM Ret_B
VAR
END_VAR
;
END_PROGRAM

(* POU Auto/Sealing_Unit, ST *)
PROGRAM Sealing_Unit
VAR
	sealingCon: INT;
	CTU_SealingConeCount: CTU;
	TON_SealingConOffDly: TON;
	CTU_SealingRevConeCount: CTU;
	TON_SealConeMissTmr: TON;
	SealUnit: INT;
	TON_SealingPisDly: TON;
	TON_SealingDly_Auto: TON;

	bASealingConeRevCountEnable: BOOL;
END_VAR
CASE sealingCon OF

0:	IF IntAllOver AND  bABagModeSelected  AND NOT bPauseSeq THEN  sealingCon:=sealingCon+1;
	ELSIF IntAllOver AND  bABoxModeSelected  AND NOT bPauseSeq THEN  sealingCon:=sealingCon+1;
	END_IF

1:	IF bABagModeSelected  AND NOT bPauseSeq THEN  bASealingConRdy_Bag:=TRUE; sealingCon:=sealingCon+1;
	ELSIF bABoxModeSelected  AND NOT bPauseSeq THEN bASealingConRdy_Box:=TRUE; sealingCon:=sealingCon+1;
	END_IF

2:	IF bABagModeSelected AND NOT bPauseSeq AND bASealingUnitOperationCom AND
	(bABagUnitRdy_243 OR bABagOperationComplete)  THEN sealingCon:=sealingCon+1;
	ELSIF bABoxModeSelected  AND NOT bPauseSeq AND bASealingUnitOperationCom AND
	(bABoxUnitRdy OR bABoxOperationCom) THEN sealingCon:=sealingCon+1;
	END_IF

3:	IF bABagModeSelected AND NOT bPauseSeq AND NOT bASealConeSet1Completed THEN
	bQASealingConFwd1:=TRUE;bASealConeSet1Started:=TRUE;bABagUnitRdy_243:=FALSE;bABagOperationComplete:=FALSE;sealingCon:=sealingCon+1;
	ELSIF bABagModeSelected AND NOT bPauseSeq AND  bASealConeSet1Completed THEN
	bQASealingConFwd2:=TRUE;bASealConeSet2Started:=TRUE;bASealConeSet1Completed:=FALSE;
	bABagUnitRdy_243:=FALSE;bABagOperationComplete:=FALSE;sealingCon:=sealingCon+1;
	ELSIF bABoxModeSelected  AND NOT bPauseSeq THEN
	bQASealingConRev:=TRUE;bABoxUnitRdy:=FALSE;bABoxOperationCom:=FALSE;sealingCon:=sealingCon+3;
	END_IF

4:	IF CTU_SealingConeCount.CV >=2 AND bABagModeSelected AND bQASealingConFwd1 THEN
	sealingCon:=sealingCon+1;
	ELSIF CTU_SealingConeCount.CV >=1 AND bABagModeSelected AND bQASealingConFwd2 THEN
	bQABagRowHolderpiston:=TRUE;sealingCon:=sealingCon+1;
	END_IF

5:	TON_SealingConOffDly(IN:=TRUE , PT:=t#2s , Q=> , ET=> );
	IF TON_SealingConOffDly.Q AND bQASealingConFwd1  THEN
	bQASealingConFwd1:=FALSE;bASealConeSet1Completed:=TRUE;sealingCon:=sealingCon+1;
	ELSIF TON_SealingConOffDly.Q AND bQASealingConFwd2  THEN
	bQASealingConFwd2:=FALSE;bASealConeSet2Completed:=FALSE;bQABagRowHolderpiston:=FALSE;
	bASealConeSet2Completed:=TRUE;sealingCon:=sealingCon+3;
	END_IF

6: 	sealingCon:=sealingCon+1;

7:	IF CTU_SealingRevConeCount.CV >= 2 AND bABoxModeSelected AND bQASealingConRev THEN
	bQASealingConRev:=FALSE;bASealConeRevSetCompleted:=TRUE;sealingCon:=sealingCon+1;END_IF

8:	sealingCon:=1;

	END_CASE

TON_SealConeMissTmr(IN:=(bQASealingConFwd1 OR bQASealingConFwd2 OR bQASealingConRev) , PT:=t#10s , Q=> , ET=> );
IF TON_SealConeMissTmr.Q AND bQASealingConFwd1 THEN bASealConeMissError1:=TRUE;
ELSIF TON_SealConeMissTmr.Q AND bQASealingConFwd2 THEN bASealConeMissError2:=TRUE;
ELSIF TON_SealConeMissTmr.Q AND bQASealingConRev THEN bASealConeMissError3:=TRUE;
END_IF

IF bASealConeMissError1 OR bASealConeMissError2 OR bASealConeMissError3 THEN
bASealConeMissError:=TRUE;bASealConeMissErrorStatus:='Cone Miss In Sealing Conveyor';END_IF

IF bASealConeMissError1 AND bQASealingConFwd1 THEN 	bQASealingConFwd1:=FALSE;
ELSIF bASealConeMissError2 AND bQASealingConFwd2 THEN 	bQASealingConFwd2:=FALSE;
ELSIF bASealConeMissError3 AND bQASealingConRev THEN 	bQASealingConRev:=FALSE;END_IF


IF bASealConeMissError1 AND NOT bPauseSeq AND bErrorReset THEN
	bASealConeMissError1:=FALSE;bQASealingConFwd1:=TRUE;
ELSIF bASealConeMissError2 AND NOT bPauseSeq AND bErrorReset THEN
	bASealConeMissError2:=FALSE;bQASealingConFwd2:=TRUE;
ELSIF bASealConeMissError3 AND NOT bPauseSeq AND bErrorReset THEN
	bASealConeMissError3:=FALSE;bQASealingConRev:=TRUE;
END_IF






IF (bQASealingConFwd1 OR bQASealingConFwd2) AND bIConeCountsensor THEN
	bASealingConeCountEnable:=TRUE;
ELSE bASealingConeCountEnable:=FALSE;END_IF
CTU_SealingConeCount(
	CU:=bASealingConeCountEnable ,
	RESET:= ,
	PV:= ,
	Q=> ,
	CV=> );

IF bQASealingConRev  AND bISpare4 THEN
	bASealingConeRevCountEnable:=TRUE;
ELSE bASealingConeRevCountEnable:=FALSE;END_IF
CTU_SealingRevConeCount(
	CU:=bASealingConeRevCountEnable ,
	RESET:= ,
	PV:= ,
	Q=> , 
	CV=> );


CASE SealUnit OF

0:	IF IntAllOver  AND NOT bPauseSeq AND bASealingUnitInt THEN
	SealUnit:=SealUnit+1;END_IF

1:	SealUnit:=SealUnit+1;

2:	IF bASealUnitStart AND NOT bPauseSeq AND bAutoModeOn  AND WrappingSafety THEN
	bQASealingSeparatorYAxisPiston:=TRUE;SealUnit:=SealUnit+1;END_IF

3:	IF bISealingSeparatorYAxisPistoEnd AND NOT bPauseSeq THEN
	bQASealingTopPiston:=TRUE;bQASealingBottomPiston:=TRUE;SealUnit:=SealUnit+1;END_IF

4:	TON_SealingPisDly(IN:=TRUE , PT:=t#2s , Q=> , ET=> );
	IF (bISealingTopPistonEnd AND bISealingBottomPistonEnd) OR TON_SealingPisDly.Q THEN
	SealUnit:=SealUnit+1;END_IF

5:	TON_SealingDly_Auto(IN:=TRUE , PT:= t#2s, Q=> , ET=> );
	IF TON_SealingDly_Auto.Q THEN SealUnit:=SealUnit+1;END_IF

6:	bQASealingSeparatorXAxisPiston:=TRUE;TON_SealingPisDly(IN:=FALSE);TON_SealingDly_Auto(IN:=FALSE);
	SealUnit:=SealUnit+1;

7:	IF bISealingSeparatorXAxisPistonEnd AND NOT bPauseSeq THEN
	bQASealingSeparatorYAxisPiston:=FALSE;
	bQASealingTopPiston:=FALSE;bQASealingBottomPiston:=FALSE;
	bQASealingSeparatorXAxisPiston:=FALSE;SealUnit:=SealUnit+1;END_IF

8:	IF SealingSafety AND NOT bPauseSeq THEN
	bASealingUnitOperationCom:=TRUE;SealUnit:=SealUnit+1;END_IF

9:	SealUnit:=0;

END_CASE
END_PROGRAM

(* POU Auto/Tilting_Piston, ST *)
PROGRAM Tilting_Piston
VAR
	TiltPis: INT;

END_VAR
CASE TiltPis OF

0: IF IntAllOver  AND NOT bPauseSeq AND bAConeFwdRevRdy THEN
	TiltPis:=TiltPis+1;END_IF

1:	TiltPis:=TiltPis+1;

2:	IF Cone1Reached  AND NOT bPauseSeq AND bIForwardPistonHome AND bIReversePistonHome THEN
	bAConeTiltingCount:=bAConeTiltingCount+1;bATiltingPistonOn:=TRUE;END_IF

3: 	IF bITiltingEnd AND NOT bPauseSeq AND NOT bAConeTiltingPistonEndRsError THEN
	Cone1Reached:=FALSE;TiltPis:=TiltPis+1;END_IF

4:	IF Cone2Reached AND  NOT bPauseSeq THEN
	bAConeTiltingCount:=bAConeTiltingCount+1;bAFwdRevPisRdy:=TRUE;Cone2Reached:=FALSE;TiltPis:=TiltPis+1;END_IF

5:	IF bAFwdRevCom AND NOT bPauseSeq THEN
	bATiltingPistonOn:=FALSE;TiltPis:=TiltPis+1;END_IF

6:	IF bITiltingHome AND NOT bPauseSeq AND NOT bAConeTiltingPistonHomeRsError THEN
	bATiltingCylCom:=TRUE;TiltPis:=TiltPis+1;END_IF

7: IF bAConeTiltingCount >= TotalNoOfCones THEN bAConeTiltingCount := 0;
	ELSE TiltPis:=TiltPis+1;END_IF

8:	TiltPis:=1;

END_CASE

IF bMcStopEnable1 OR NOT bAutoModeOn  THEN
TiltPis:=0;bAConeTiltingCount := 0;bATiltingCylCom:=FALSE;
bAFwdRevPisRdy:=FALSE;Cone2Reached:=FALSE;Cone1Reached:=FALSE;
bATiltingPistonOn:=FALSE;bAConeFwdRevRdy:=FALSE;END_IF
END_PROGRAM

(* POU Auto/Wrapping_Unit, ST *)
PROGRAM Wrapping_Unit
VAR
	WrappingCon: INT;
	WrapPis: INT;

	bASealConRdy: BOOL;
END_VAR
CASE WrappingCon OF
0: 	IF IntAllOver  AND NOT bPauseSeq AND bAWrappingPisCylComInt THEN
	WrappingCon:=WrappingCon+1;END_IF

1:	IF (bAWrappingPisCylCom OR bAWrappingPisCylComInt ) AND NOT bPauseSeq THEN
	bAWrappingConRdy:=FALSE;bAWrappingPisCylCom:=FALSE;
	bAWrappingPisCylComInt:=FALSE;WrappingCon:=WrappingCon+1;END_IF

2:	IF bAWrappingConRdy AND WrappingSafety AND NOT bIWrappingCone1 AND NOT bIWrappingCone2 AND NOT bPauseSeq THEN
	bAWrapConeAlaignError:=FALSE;bAWrappingConRdy:=FALSE;
	sWrappingConStatus:='Continue Machine Runnig';WrappingCon:=WrappingCon+2;

	ELSIF bAWrappingConRdy AND WrappingSafety AND NOT bPauseSeq AND bIWrappingCone1  THEN
	bAWrapConeAlaignError:=TRUE;sWrappingConStatus:='Please Check Wrap Cone 1';WrappingCon:=WrappingCon+1;

	ELSIF bAWrappingConRdy AND WrappingSafety AND NOT bPauseSeq AND bIWrappingCone2  THEN
	bAWrapConeAlaignError:=TRUE;sWrappingConStatus:='Please Check Wrap Cone 2';WrappingCon:=WrappingCon+1;

	ELSIF bAWrappingConRdy AND WrappingSafety AND NOT bPauseSeq AND (bIWrappingCone1 OR bIWrappingCone2)  THEN
	bAWrapConeAlaignError:=TRUE;sWrappingConStatus:='Please Check Wrap Cone 1 & 2';WrappingCon:=WrappingCon+1;
	END_IF

3:	IF bErrorReset AND NOT bIWrappingCone1 AND NOT bIWrappingCone2 AND NOT bPauseSeq THEN
	bAWrapConeAlaignError:=FALSE;sWrappingConStatus:='Continue Machine Runnig';WrappingCon:=WrappingCon+1;END_IF

4:	bAWrappingConOn:=TRUE;WrappingCon:=WrappingCon+1;

5:	IF bIWrappingCone1 AND bIWrappingCone2 THEN
	bAWrappingConOn:=FALSE;WrappingCon:=WrappingCon+1;END_IF

6:	IF NOT bAWrapConeAlaignError1 AND NOT bPauseSeq THEN
	bAWrappingPisRdy:=TRUE;bASealConRdy:=TRUE;WrappingCon:=WrappingCon+1;END_IF

7:	WrappingCon:=1;

END_CASE

CASE WrapPis OF
0:	IF bAWrappingPisRdy AND NOT bPauseSeq THEN
	bAWrapPiston1On:=TRUE;bAWrapPiston2On:=TRUE;WrapPis:=WrapPis+1;END_IF

1:	bAWrappingPisRdy:=FALSE;WrapPis:=WrapPis+1;

2:	IF bIWrappingChanelPiston1Middle OR bIWrappingChanelPiston2Middle THEN
	WrapPis:=WrapPis+1;END_IF

3:	IF bASealingConRdy AND NOT bPauseSeq THEN
	WrapPis:=WrapPis+2;
	ELSIF NOT bASealingConRdy THEN
	 bAWrapPiston1On:=FALSE;bAWrapPiston2On:=FALSE;WrapPis:=WrapPis+1;END_IF

4:	IF bASealingConRdy AND NOT bPauseSeq THEN
	bAWrapPiston1On:=TRUE;bAWrapPiston2On:=TRUE;WrapPis:=WrapPis+1;END_IF

5: 	IF bIWrappingChanelPiston1End AND bIWrappingChanelPiston2End
	AND NOT bASheetFeedError AND NOT bAWrapPis1EndRsError AND NOT bAWrapPis2EndRsError
	AND NOT bPauseSeq THEN WrapPis:=WrapPis+1;
	 bAWrapPiston1On:=FALSE;bAWrapPiston2On:=FALSE;WrapPis:=WrapPis+1;
	ELSIF  bIWrappingChanelPiston1End AND bIWrappingChanelPiston2End AND  bASheetFeedError THEN WrapPis:=WrapPis+1;
	ELSIF bAWrapPis1EndRsError OR bAWrapPis2EndRsError THEN WrapPis:=WrapPis+1;
	END_IF

6:  	IF bErrorReset AND NOT bPauseSeq AND NOT bAWrapPis1EndRsError AND NOT bAWrapPis2EndRsError THEN
	WrapPis:=5;END_IF

7:	IF WrappingSafety AND NOT bPauseSeq THEN
	bAWrappingPisCylCom:=TRUE; bASealUnitStart:=TRUE;WrapPis:=WrapPis+1;END_IF

8:	WrapPis:=0;

END_CASE
END_PROGRAM

(* POU DataLog/ErrorData_Report, ST *)
PROGRAM ErrorData_Report
VAR
END_VAR
;
END_PROGRAM

(* POU DataLog/Print_Report, ST *)
PROGRAM Print_Report
VAR
	step: INT;


	TON_2: TON;
	TON_1: TON;
END_VAR
IF PrintEnable_TogHmi THEN PrintEnabled:=TRUE;PrintValue:=1;ELSE PrintEnabled:=FALSE;PrintValue:=0;END_IF

		ProductionData_PrintData.Print						:=INT_TO_STRING( PrintValue );
		ProductionData_PrintData.ConeType1				:=(COUNT_DIS);
		ProductionData_PrintData.Blend1					:=(BLEND_DIS);
		ProductionData_PrintData.DefaultnetWt1				:=(Actual_NetWeight_Report);
		ProductionData_PrintData.DefaultGrossWt1			:=(Actual_GrossWeight_Report);
		ProductionData_PrintData.LotNo1					:=(LOTNO_DIS);
		ProductionData_PrintData.BagNo1					:=DINT_TO_STRING(CARTONNO_DIS);
		ProductionData_PrintData.Shade1					:=(SHADE_DIS);

		(*	######## Print Data Values		#####	*)

ProductionDataValues_Print:= CONCAT(ProductionData_PrintData.Print,',');
ProductionDataValues_Print:=	 CONCAT( ProductionDataValues_Print,ProductionData_PrintData.ConeType1);
ProductionDataValues_Print:= CONCAT( ProductionDataValues_Print,',');
ProductionDataValues_Print:=	 CONCAT( ProductionDataValues_Print,ProductionData_PrintData.Blend1);
ProductionDataValues_Print:= CONCAT( ProductionDataValues_Print,',');
ProductionDataValues_Print:=	 CONCAT( ProductionDataValues_Print,ProductionData_PrintData.DefaultnetWt1);
ProductionDataValues_Print:= CONCAT( ProductionDataValues_Print,',');
ProductionDataValues_Print:=	 CONCAT( ProductionDataValues_Print,ProductionData_PrintData.DefaultGrossWt1);
ProductionDataValues_Print:= CONCAT( ProductionDataValues_Print,',');
ProductionDataValues_Print:=	 CONCAT( ProductionDataValues_Print,ProductionData_PrintData.LotNo1);
ProductionDataValues_Print:= CONCAT( ProductionDataValues_Print,',');
ProductionDataValues_Print:=	 CONCAT( ProductionDataValues_Print,ProductionData_PrintData.BagNo1);
ProductionDataValues_Print:= CONCAT( ProductionDataValues_Print,',');
ProductionDataValues_Print:=	 CONCAT( ProductionDataValues_Print,ProductionData_PrintData.Shade1);
ProductionDataValues_Print:= CONCAT( ProductionDataValues_Print,'$0A');


					(*	######## Print Data head#####	*)
ProductionData_Print:= CONCAT( 'Print',',');
		ProductionData_Print:=	 CONCAT( ProductionData_Print,'Count Type');
		ProductionData_Print:= CONCAT( ProductionData_Print,',');
ProductionData_Print:=	 CONCAT( ProductionData_Print,'Blend');
		ProductionData_Print:= CONCAT( ProductionData_Print,',');
ProductionData_Print:=	 CONCAT( ProductionData_Print,'NetWt');
		ProductionData_Print:= CONCAT( ProductionData_Print,',');
ProductionData_Print:=	 CONCAT( ProductionData_Print,'Grss Wt');
		ProductionData_Print:= CONCAT( ProductionData_Print,',');
ProductionData_Print:=	 CONCAT( ProductionData_Print,'Lot No');
		ProductionData_Print:= CONCAT( ProductionData_Print,',');
ProductionData_Print:=	 CONCAT( ProductionData_Print,'Bag No');
		ProductionData_Print:= CONCAT( ProductionData_Print,',');
ProductionData_Print:=	 CONCAT( ProductionData_Print,'Shade');
		ProductionData_Print:= CONCAT( ProductionData_Print,'$0A');

FB_FileOpen1(
	sNetId:='192.168.225.76.1.1',
	sPathName:= '\\ACPBAG\Reports\productiondata.csv' ,
	nMode:=FOPEN_MODEAPPEND ,
	ePath:=PATH_GENERIC ,
	bExecute:= ,
	tTimeout:=T#2s ,
	bBusy=> ,
	bError=> ,
	nErrId=> ,
	hFile=> );

FB_FileWrite1(
	sNetId:='192.168.225.76.1.1',
	hFile:=FB_FileOpen1.hFile ,
	pWriteBuff:=ADR(ProductionDataValues_Print_Com),
	cbWriteLen:=LEN(ProductionDataValues_Print_Com),
	bExecute:= ,
	tTimeout:=T#2s ,
	bBusy=> ,
	bError=> ,
	nErrId=> ,
	cbWrite=> );


FB_FileClose1(
	sNetId:='192.168.225.76.1.1',
	hFile:=FB_FileOpen1.hFile ,
	bExecute:= ,
	tTimeout:=T#2s ,
	bBusy=> ,
	bError=> ,
	nErrId=> );

FB_FileDelete1(
	sNetId:='192.168.225.76.1.1',
	sPathName:= '\\ACPBAG\Reports\productiondata.csv' ,
	ePath:=PATH_GENERIC ,
	bExecute:= ,
	tTimeout:=T#2s ,
	bBusy=> ,
	bError=> ,
	nErrId=> );

CASE step OF

0: IF PrintOk THEN
	TON_2(IN:=FALSE);
	FB_FileOpen1.bExecute:=TRUE;
	IF NOT FB_FileOpen1.bBusy AND NOT FB_FileOpen1.bError AND FB_FileOpen1.hFile>0 THEN  step:=step+1;END_IF
	END_IF

1:	IF NOT FB_FileOpen1.bBusy AND NOT FB_FileOpen1.bError AND FB_FileOpen1.hFile>0 THEN  PrintOk:=FALSE;step:=step+1;END_IF

2:
	ProductionDataValues_Print_Com:=ProductionData_Print;
	FB_FileWrite1.bExecute:=TRUE;
	IF NOT FB_FileWrite1.bBusy AND NOT FB_FileWrite1.bError THEN step:=step+1;END_IF

3:	IF NOT FB_FileWrite1.bBusy AND NOT FB_FileWrite1.bError THEN FB_FileWrite1.bExecute:=FALSE; step:=step+1;END_IF

4:	ProductionDataValues_Print_Com:=ProductionDataValues_Print;
	FB_FileWrite1.bExecute:=TRUE;
	IF NOT FB_FileWrite1.bBusy AND NOT FB_FileWrite1.bError THEN step:=step+1;END_IF

5:	step:=step+1;

6:	IF NOT FB_FileWrite1.bBusy AND NOT FB_FileWrite1.bError THEN FB_FileWrite1.bExecute:=FALSE; step:=step+1;END_IF


7:	FB_FileClose1.bExecute:=TRUE;
	 IF NOT FB_FileClose1.bBusy AND NOT FB_FileClose1.bError THEN  step:=step+1;END_IF

8:	TON_1(IN:=TRUE , PT:=t#0.1s , Q=> , ET=> );
	IF TON_1.Q THEN step:=step+1;END_IF

9:	IF NOT FB_FileDelete1.bBusy AND NOT FB_FileDelete1.bError THEN
	TON_1(IN:=FALSE);
	(*FB_FileDelete1.bExecute:=TRUE;*)step:=step+1;END_IF

10:
	FB_FileOpen1.bExecute:=FALSE;
	FB_FileWrite1.bExecute:=FALSE;
	FB_FileClose1.bExecute:=FALSE;
	FB_FileDelete1.bExecute:=FALSE;
	step:=step+1;

11:		TON_2(IN:=TRUE , PT:=t#10s , Q=> , ET=> );
	IF TON_2.Q THEN(* PrintOk:=TRUE;	*) step:=0;END_IF

END_CASE
END_PROGRAM

(* POU Print, ST *)
PROGRAM Print
VAR

	step: INT;


	TON_2: TON;
	TON_1: TON;
END_VAR
IF PrintEnable_TogHmi THEN PrintEnabled:=TRUE;PrintValue:=1;ELSE PrintEnabled:=FALSE;PrintValue:=0;END_IF

		ProductionData_PrintData.Print						:=INT_TO_STRING( PrintValue );
		ProductionData_PrintData.ConeType1				:=(COUNT_DIS);
		ProductionData_PrintData.Blend1					:=(BLEND_DIS);
		ProductionData_PrintData.DefaultnetWt1				:=(Actual_NetWeight_Report);
		ProductionData_PrintData.DefaultGrossWt1			:=(Actual_GrossWeight_Report);
		ProductionData_PrintData.LotNo1					:=(LOTNO_DIS);
		ProductionData_PrintData.BagNo1					:=DINT_TO_STRING(CARTONNO_DIS);
		ProductionData_PrintData.Shade1					:=(SHADE_DIS);

		(*	######## Print Data Values		#####	*)

ProductionDataValues_Print:= CONCAT(ProductionData_PrintData.Print,',');
ProductionDataValues_Print:=	 CONCAT( ProductionDataValues_Print,ProductionData_PrintData.ConeType1);
ProductionDataValues_Print:= CONCAT( ProductionDataValues_Print,',');
ProductionDataValues_Print:=	 CONCAT( ProductionDataValues_Print,ProductionData_PrintData.Blend1);
ProductionDataValues_Print:= CONCAT( ProductionDataValues_Print,',');
ProductionDataValues_Print:=	 CONCAT( ProductionDataValues_Print,ProductionData_PrintData.DefaultnetWt1);
ProductionDataValues_Print:= CONCAT( ProductionDataValues_Print,',');
ProductionDataValues_Print:=	 CONCAT( ProductionDataValues_Print,ProductionData_PrintData.DefaultGrossWt1);
ProductionDataValues_Print:= CONCAT( ProductionDataValues_Print,',');
ProductionDataValues_Print:=	 CONCAT( ProductionDataValues_Print,ProductionData_PrintData.LotNo1);
ProductionDataValues_Print:= CONCAT( ProductionDataValues_Print,',');
ProductionDataValues_Print:=	 CONCAT( ProductionDataValues_Print,ProductionData_PrintData.BagNo1);
ProductionDataValues_Print:= CONCAT( ProductionDataValues_Print,',');
ProductionDataValues_Print:=	 CONCAT( ProductionDataValues_Print,ProductionData_PrintData.Shade1);
ProductionDataValues_Print:= CONCAT( ProductionDataValues_Print,'$0A');


					(*	######## Print Data head#####	*)
ProductionData_Print:= CONCAT( 'Print',',');
		ProductionData_Print:=	 CONCAT( ProductionData_Print,'Count Type');
		ProductionData_Print:= CONCAT( ProductionData_Print,',');
ProductionData_Print:=	 CONCAT( ProductionData_Print,'Blend');
		ProductionData_Print:= CONCAT( ProductionData_Print,',');
ProductionData_Print:=	 CONCAT( ProductionData_Print,'NetWt');
		ProductionData_Print:= CONCAT( ProductionData_Print,',');
ProductionData_Print:=	 CONCAT( ProductionData_Print,'Grss Wt');
		ProductionData_Print:= CONCAT( ProductionData_Print,',');
ProductionData_Print:=	 CONCAT( ProductionData_Print,'Lot No');
		ProductionData_Print:= CONCAT( ProductionData_Print,',');
ProductionData_Print:=	 CONCAT( ProductionData_Print,'Bag No');
		ProductionData_Print:= CONCAT( ProductionData_Print,',');
ProductionData_Print:=	 CONCAT( ProductionData_Print,'Shade');
		ProductionData_Print:= CONCAT( ProductionData_Print,'$0A');

FB_FileOpen1(
	sNetId:='192.168.225.76.1.1',
	sPathName:= '\\ACPBAG\Reports\productiondata.csv' ,
	nMode:=FOPEN_MODEAPPEND ,
	ePath:=PATH_GENERIC ,
	bExecute:= ,
	tTimeout:=T#2s ,
	bBusy=> ,
	bError=> ,
	nErrId=> ,
	hFile=> );

FB_FileWrite1(
	sNetId:='192.168.225.76.1.1',
	hFile:=FB_FileOpen1.hFile ,
	pWriteBuff:=ADR(ProductionDataValues_Print_Com),
	cbWriteLen:=LEN(ProductionDataValues_Print_Com),
	bExecute:= ,
	tTimeout:=T#2s ,
	bBusy=> ,
	bError=> ,
	nErrId=> ,
	cbWrite=> );


FB_FileClose1(
	sNetId:='192.168.225.76.1.1',
	hFile:=FB_FileOpen1.hFile ,
	bExecute:= ,
	tTimeout:=T#2s ,
	bBusy=> ,
	bError=> ,
	nErrId=> );

FB_FileDelete1(
	sNetId:='192.168.225.76.1.1',
	sPathName:= '\\ACPBAG\Reports\productiondata.csv' ,
	ePath:=PATH_GENERIC ,
	bExecute:= ,
	tTimeout:=T#2s ,
	bBusy=> ,
	bError=> ,
	nErrId=> );

CASE step OF

0: IF PrintOk THEN
	TON_2(IN:=FALSE);
	FB_FileOpen1.bExecute:=TRUE;
	IF NOT FB_FileOpen1.bBusy AND NOT FB_FileOpen1.bError AND FB_FileOpen1.hFile>0 THEN  step:=step+1;END_IF
	END_IF

1:	IF NOT FB_FileOpen1.bBusy AND NOT FB_FileOpen1.bError AND FB_FileOpen1.hFile>0 THEN  PrintOk:=FALSE;step:=step+1;END_IF

2:
	ProductionDataValues_Print_Com:=ProductionData_Print;
	FB_FileWrite1.bExecute:=TRUE;
	IF NOT FB_FileWrite1.bBusy AND NOT FB_FileWrite1.bError THEN step:=step+1;END_IF

3:	IF NOT FB_FileWrite1.bBusy AND NOT FB_FileWrite1.bError THEN FB_FileWrite1.bExecute:=FALSE; step:=step+1;END_IF

4:	ProductionDataValues_Print_Com:=ProductionDataValues_Print;
	FB_FileWrite1.bExecute:=TRUE;
	IF NOT FB_FileWrite1.bBusy AND NOT FB_FileWrite1.bError THEN step:=step+1;END_IF

5:	step:=step+1;

6:	IF NOT FB_FileWrite1.bBusy AND NOT FB_FileWrite1.bError THEN FB_FileWrite1.bExecute:=FALSE; step:=step+1;END_IF


7:	FB_FileClose1.bExecute:=TRUE;
	 IF NOT FB_FileClose1.bBusy AND NOT FB_FileClose1.bError THEN  step:=step+1;END_IF

8:	TON_1(IN:=TRUE , PT:=t#0.1s , Q=> , ET=> );
	IF TON_1.Q THEN step:=step+1;END_IF

9:	IF NOT FB_FileDelete1.bBusy AND NOT FB_FileDelete1.bError THEN
	TON_1(IN:=FALSE);
	(*FB_FileDelete1.bExecute:=TRUE;*)step:=step+1;END_IF

10:
	FB_FileOpen1.bExecute:=FALSE;
	FB_FileWrite1.bExecute:=FALSE;
	FB_FileClose1.bExecute:=FALSE;
	FB_FileDelete1.bExecute:=FALSE;
	step:=step+1;

11:		TON_2(IN:=TRUE , PT:=t#10s , Q=> , ET=> );
	IF TON_2.Q THEN(* PrintOk:=TRUE;	*) step:=0;END_IF

END_CASE
END_PROGRAM

(* POU DataLog/ProductionData_Report, ST *)
PROGRAM ProductionData_Report
VAR

	TON_Indo1: TON;
	TON_Indo2: TON;
	TON_Indo3: TON;
	TON_Indo4: TON;
	TON_Newdaydly: TON;
	TON_NEWDAY: TON;
	TON_NewdaydlyError: TON;
	TON_writedly: TON;
	TON_Opendly: TON;
END_VAR
	ProductionData_ReportData1.SERIALNO	:=DINT_TO_STRING(SerialNo);
		ProductionData_ReportData1.SDATE	:=(wTodayToHmiFinal);
		ProductionData_ReportData1.BAGNO	:=DINT_TO_STRING(CARTONNO_DIS);
		ProductionData_ReportData1.COUNTCODE	:=(COUNT_DIS);
		ProductionData_ReportData1.LOTNO	:=(LOTNO_DIS);
		ProductionData_ReportData1.DFLTNETWEIGHT	:=(Default_NetWeight_Report);
		ProductionData_ReportData1.ACTNETWEIGHT	:=(Actual_NetWeight_Report);



FB_FileOpen_Indo(
	sNetId:='192.168.225.76.1.1',
	sPathName:= ReportPath_Final_2,
	nMode:=FOPEN_MODEAPPEND ,
	ePath:=PATH_GENERIC ,
	bExecute:= ,
	tTimeout:=T#2s ,
	bBusy=> ,
	bError=> ,
	nErrId=> ,
	hFile=> );

FB_FileWrite_Indo(
	sNetId:='192.168.225.76.1.1',
	hFile:=FB_FileOpen_Indo.hFile ,
	pWriteBuff:=ADR(ProductionDataValues_IndoPrint_Com),
	cbWriteLen:=LEN(ProductionDataValues_IndoPrint_Com),
	bExecute:= ,
	tTimeout:=T#2s ,
	bBusy=> ,
	bError=> ,
	nErrId=> ,
	cbWrite=> );


FB_FileClose_Indo(
	sNetId:='192.168.225.76.1.1',
	hFile:=FB_FileOpen_Indo.hFile ,
	bExecute:= ,
	tTimeout:=T#2s ,
	bBusy=> ,
	bError=> ,
	nErrId=> );

FB_FileDelete_Indo(
	sNetId:='192.168.225.76.1.1',
	sPathName:= ReportPath_Final_2,
	ePath:=PATH_GENERIC ,
	bExecute:= ,
	tTimeout:=T#2s ,
	bBusy=> ,
	bError=> ,
	nErrId=> );

R_TRIG_IndoPrint(CLK:=( bANewDay OR testbit)  , Q=> );

CASE IndoReport OF
0:	  IF TON_NEWDAY.Q   THEN	sOldDay := sDay;TON_Newdaydly(IN:=TRUE , PT:=t#0.2s , Q=> , ET=> );
		IF TON_Newdaydly.Q THEN
		bANewDay:=FALSE;IndoReport:=1; SerialNo:=1;FB_FileOpen_Indo.bExecute:=TRUE;END_IF END_IF

1:	TON_Newdaydly(IN:=FALSE);TON_NEWDAY(IN:=FALSE);
	IF NOT FB_FileOpen_Indo.bBusy AND NOT FB_FileOpen_Indo.bError AND FB_FileOpen_Indo.hFile>0 THEN ReportHead1_Indo:=TRUE;END_IF

	IF ReportHead1_Indo THEN
	ProductionData_IndoPrint:= CONCAT( 'SL NO',',');
	ProductionData_IndoPrint:=	 CONCAT( ProductionData_IndoPrint,'DATE/TIME');
		ProductionData_IndoPrint:= CONCAT( ProductionData_IndoPrint,',');
	ProductionData_IndoPrint:=	 CONCAT( ProductionData_IndoPrint,'BAG NO');
		ProductionData_IndoPrint:= CONCAT( ProductionData_IndoPrint,',');
	ProductionData_IndoPrint:=	 CONCAT( ProductionData_IndoPrint,'COUNT');
		ProductionData_IndoPrint:=CONCAT( ProductionData_IndoPrint,',');
	ProductionData_IndoPrint:=	 CONCAT( ProductionData_IndoPrint,'LOT NO');
		ProductionData_IndoPrint:=CONCAT( ProductionData_IndoPrint,',');
	ProductionData_IndoPrint:=	 CONCAT( ProductionData_IndoPrint,'DFLT NET WT');
		ProductionData_IndoPrint:=CONCAT( ProductionData_IndoPrint,',');
	ProductionData_IndoPrint:=	 CONCAT( ProductionData_IndoPrint,'ACT NET WT');
		ProductionData_IndoPrint:= CONCAT( ProductionData_IndoPrint,'$0A');
	IndoReport:=7; END_IF

2:	PROCESSCOMPLETE:=FALSE;ReportHead1_Indo:=FALSE;ProductionDataValues_IndoPrint_Com:=ProductionData_IndoPrint;
	TON_Indo1(IN:=TRUE , PT:=t#5s , Q=> , ET=> );
	FB_FileWrite_Indo.bExecute:=TRUE;
	IF NOT FB_FileWrite_Indo.bBusy AND NOT FB_FileWrite_Indo.bError AND FB_FileWrite_Indo.hFile>0 AND TON_Indo1.Q THEN IndoReport:=IndoReport+1; END_IF

3:	ProductionDataValues_IndoPrint_Com:=ProductionData_IndoPrint;
	FB_FileWrite_Indo.bExecute:=TRUE;
	IF NOT FB_FileWrite_Indo.bBusy AND NOT FB_FileWrite_Indo.bError THEN IndoReport:=IndoReport+1; END_IF

4:	FB_FileWrite_Indo.bExecute:=FALSE;ProductionData_IndoPrint:='';IndoReport:=IndoReport+1;

5:	ReportHead2_Indo:=TRUE;
	IF ReportHead2_Indo THEN IndoReport:=IndoReport+1;END_IF

6:	ProductionData_IndoPrint:=	 CONCAT( ProductionData_IndoPrint,'Cn13Wt');
		ProductionData_IndoPrint:=CONCAT( ProductionData_IndoPrint,',');
	ProductionData_IndoPrint:=	 CONCAT( ProductionData_IndoPrint,'Cn14Wt');
		ProductionData_IndoPrint:=CONCAT( ProductionData_IndoPrint,',');
	ProductionData_IndoPrint:=	 CONCAT( ProductionData_IndoPrint,'Cn15Wt');
		ProductionData_IndoPrint:=CONCAT( ProductionData_IndoPrint,',');
	ProductionData_IndoPrint:=	 CONCAT( ProductionData_IndoPrint,'Cn16Wt');
		ProductionData_IndoPrint:=CONCAT( ProductionData_IndoPrint,',');
	ProductionData_IndoPrint:=	 CONCAT( ProductionData_IndoPrint,'Cn17Wt');
		ProductionData_IndoPrint:=CONCAT( ProductionData_IndoPrint,',');
	ProductionData_IndoPrint:=	 CONCAT( ProductionData_IndoPrint,'Cn18Wt');
		ProductionData_IndoPrint:=CONCAT( ProductionData_IndoPrint,',');
	ProductionData_IndoPrint:=	 CONCAT( ProductionData_IndoPrint,'Cn19Wt');
		ProductionData_IndoPrint:=CONCAT( ProductionData_IndoPrint,',');
	ProductionData_IndoPrint:=	 CONCAT( ProductionData_IndoPrint,'Cn20Wt');
		ProductionData_IndoPrint:=CONCAT( ProductionData_IndoPrint,',');
	ProductionData_IndoPrint:=	 CONCAT( ProductionData_IndoPrint,'Cn21Wt');
		ProductionData_IndoPrint:=CONCAT( ProductionData_IndoPrint,',');
	ProductionData_IndoPrint:=	 CONCAT( ProductionData_IndoPrint,'Cn22Wt');
		ProductionData_IndoPrint:=CONCAT( ProductionData_IndoPrint,',');
	ProductionData_IndoPrint:=	 CONCAT( ProductionData_IndoPrint,'Cn23Wt');
		ProductionData_IndoPrint:=CONCAT( ProductionData_IndoPrint,',');
	ProductionData_IndoPrint:=	 CONCAT( ProductionData_IndoPrint,'Cn24Wt');
		ProductionData_IndoPrint:= CONCAT( ProductionData_IndoPrint,'$0A');
	ReportHead2_Indo:=FALSE;
	IndoReport:=IndoReport+1;

7:	ReportHead1_Indo:=FALSE;ProductionDataValues_IndoPrint_Com:=ProductionData_IndoPrint;
	TON_Indo2(IN:=TRUE , PT:=t#5s , Q=> , ET=> );
	FB_FileWrite_Indo.bExecute:=TRUE;
	IF NOT FB_FileWrite_Indo.bBusy AND NOT FB_FileWrite_Indo.bError  AND TON_Indo2.Q THEN  IndoReport:=IndoReport+1; END_IF

8:	FB_FileWrite_Indo.bExecute:=FALSE;
	FB_FileClose_Indo.bExecute:=TRUE;
	 IF NOT FB_FileClose_Indo.bBusy AND NOT FB_FileClose_Indo.bError THEN FB_FileOpen_Indo.bExecute:=FALSE; IndoReport:=IndoReport+1;END_IF(*ProductionData_IndoPrint:='';*)

9:	FB_FileClose_Indo.bExecute:=FALSE;
	IF ReportSave OR testbit THEN

	FB_FileOpen_Indo.bExecute:=TRUE;
	IF NOT FB_FileOpen_Indo.bBusy AND NOT FB_FileOpen_Indo.bError AND FB_FileOpen_Indo.hFile>0 THEN
	ReportBot1_Indo:=TRUE;END_IF

	IF ReportBot1_Indo THEN IndoReport:=IndoReport+1;END_IF END_IF

10:
	ProductionData_IndoPrint2:= CONCAT(ProductionData_ReportData1.SERIALNO,',');
	ProductionData_IndoPrint2:=	 CONCAT( ProductionData_IndoPrint2,ProductionData_ReportData1.SDATE	);
		ProductionData_IndoPrint2:= CONCAT( ProductionData_IndoPrint2,',');
	ProductionData_IndoPrint2:=	 CONCAT( ProductionData_IndoPrint2,ProductionData_ReportData1.BAGNO	);
		ProductionData_IndoPrint2:= CONCAT( ProductionData_IndoPrint2,',');
	ProductionData_IndoPrint2:=	 CONCAT( ProductionData_IndoPrint2,ProductionData_ReportData1.COUNTCODE);
		ProductionData_IndoPrint2:= CONCAT( ProductionData_IndoPrint2,',');
	ProductionData_IndoPrint2:=	 CONCAT( ProductionData_IndoPrint2,ProductionData_ReportData1.LOTNO);
		ProductionData_IndoPrint2:= CONCAT( ProductionData_IndoPrint2,',');
	ProductionData_IndoPrint2:=	 CONCAT( ProductionData_IndoPrint2,ProductionData_ReportData1.DFLTNETWEIGHT);
		ProductionData_IndoPrint2:= CONCAT( ProductionData_IndoPrint2,',');
	ProductionData_IndoPrint2:=	 CONCAT( ProductionData_IndoPrint2,ProductionData_ReportData1.ACTNETWEIGHT);
		ProductionData_IndoPrint2:= CONCAT( ProductionData_IndoPrint2,'$0A');
	ReportBot1_Indo:=FALSE;ReportSave:=FALSE;
	IndoReport:=15;


11:	ProductionDataValues_IndoPrint_Com:=ProductionData_IndoPrint2;
	TON_Indo3(IN:=TRUE , PT:=t#5s , Q=> , ET=> );
	FB_FileWrite_Indo.bExecute:=TRUE;
	IF NOT FB_FileWrite_Indo.bBusy AND NOT FB_FileWrite_Indo.bError AND TON_Indo3.Q THEN
	 IndoReport:=IndoReport+1; END_IF

12:	FB_FileWrite_Indo.bExecute:=FALSE;IndoReport:=IndoReport+1;

13:	ReportBot2_Indo:=TRUE;
	IF ReportBot2_Indo THEN IndoReport:=IndoReport+1;END_IF

14:	ReportBot2_Indo:=FALSE;
	IndoReport:=IndoReport+1;

15:	ProductionDataValues_IndoPrint_Com:=ProductionData_IndoPrint2;
	TON_Indo4(IN:=TRUE , PT:=t#5s , Q=> , ET=> );
	FB_FileWrite_Indo.bExecute:=TRUE; IndoReport:=IndoReport+1;


16:	IF NOT FB_FileWrite_Indo.bBusy AND NOT FB_FileWrite_Indo.bError THEN
	FB_FileWrite_Indo.bExecute:=FALSE; IndoReport:=IndoReport+1;END_IF


17:	TON_Indo3(IN:=FALSE);TON_Indo4(IN:=FALSE);TON_Indo2(IN:=FALSE);
	TON_Indo1(IN:=FALSE);FB_FileWrite_Indo.bExecute:=FALSE;IndoReport:=IndoReport+1;

18:	FB_FileClose_Indo.bExecute:=TRUE;
	 IF NOT FB_FileClose_Indo.bBusy AND NOT FB_FileClose_Indo.bError THEN
	IndoReport:=20;END_IF

19:	IF bANewDay THEN
	IndoReport:=IndoReport+1;
	ELSIF NOT bANewDay THEN FB_FileOpen_Indo.bExecute:=FALSE; IndoReport:=9;
	END_IF

20:	FB_FileOpen_Indo.bExecute:=FALSE;SerialNo:=SerialNo+1;IndoReport:=9;
END_CASE

	IF sDay <> sOldDay THEN
	bANewDay:=TRUE;IndoReport:=0; SerialNo:=0;END_IF
	TON_NEWDAY(IN:=bANewDay , PT:=T#0.5s , Q=> , ET=> );

CASE WriteError OF

0:	IF FB_FileWrite_Indo.bError THEN
	FB_FileWrite_Indo.bExecute:=FALSE;TON_writedly(IN:=FALSE);
	WriteError:=WriteError+1;END_IF

1:	TON_writedly(IN:=TRUE , PT:=t#2s , Q=> , ET=> );
	IF TON_writedly.Q THEN
	 FB_FileWrite_Indo.bExecute:=TRUE;WriteError:=WriteError+1;END_IF

2:	TON_writedly(IN:=FALSE);WriteError:=0;

END_CASE

CASE OpenError OF

0:	IF FB_FileOpen_Indo.bError THEN
	FB_FileOpen_Indo.bExecute:=FALSE;TON_Opendly(IN:=FALSE);
	OpenError:=OpenError+1;END_IF

1:	TON_Opendly(IN:=TRUE , PT:=t#2s , Q=> , ET=> );
	IF TON_Opendly.Q THEN
	FB_FileOpen_Indo.bExecute:=TRUE;OpenError:=OpenError+1;END_IF

2:	TON_Opendly(IN:=FALSE);OpenError:=0;

END_CASE
END_PROGRAM

(* POU Initialize/Bag_Int, ST *)
PROGRAM Bag_Int
VAR
	BagUnitInt: INT;
	bQBagHolder: BOOL;
	bQRBagPusherForwardPiston: BOOL;
	bQRBagPusherReversePiston: BOOL;
	bQRBagTiltingpistonForward: BOOL;
	bQRBagTiltingpistonReverse: BOOL;
	bQRColumnStopperPiston: BOOL;
	bQRColumnReversePiston: BOOL;
	bQRBagUp_Down180piston: BOOL;
	bQRBagUp_Down50piston: BOOL;
	bQRConePusher1Piston: BOOL;
	bQABagUp_Down180piston: BOOL;
	bQAConePusher3Piston: BOOL;
	bQAColumnStopperPiston: BOOL;
	bQABagUp_Down50piston: BOOL;
	bQAConePusher1Piston: BOOL;
END_VAR
CASE BagUnitInt OF

0:	IF bRBagUnitIntRdy  AND NOT bPauseSeq AND NOT bQBagHolder THEN
	BagUnitInt:=BagUnitInt+1;END_IF

1:	IF  bIBagPusherPistonHome THEN BagUnitInt:=BagUnitInt+2;
	ELSIF NOT bIBagPusherPistonHome AND NOT bPauseSeq THEN
	bQRBagPusherForwardPiston:=FALSE;bQRBagPusherReversePiston:= TRUE;END_IF

2:	IF bIBagPusherPistonHome THEN
	bQRBagPusherReversePiston:= FALSE;bQRBagPusherForwardPiston:=FALSE;BagUnitInt:=BagUnitInt+1;END_IF

3:	bRBagUnitIntRdy:=FALSE; BagUnitInt:=BagUnitInt+1;

4:	IF bIBagTiltingPistonHome THEN BagUnitInt:=BagUnitInt+2;
	ELSIF NOT bIBagTiltingPistonHome AND NOT bPauseSeq THEN
	bQRBagTiltingpistonForward:=FALSE;bQRBagTiltingpistonReverse:=TRUE;BagUnitInt:=BagUnitInt+1;END_IF

5:	IF  bIBagTiltingPistonHome THEN
	bQRBagTiltingpistonForward:=FALSE;bQRBagTiltingpistonReverse:=FALSE;BagUnitInt:=BagUnitInt+1;END_IF

6:	bQRColumnStopperPiston:=FALSE;bQRColumnReversePiston:=FALSE;BagUnitInt:=BagUnitInt+1;

7:	IF bISeperatorPlatePistonHome AND bIConePusher1PistonHome AND NOT bQBagHolder
	AND bIBagPusherPistonHome AND bIBagTiltingPistonHome AND NOT bPauseSeq THEN
	bQRBagUp_Down180piston:=TRUE;BagUnitInt:=BagUnitInt+1;END_IF

8:	IF bIBagUpDown180PistonEnd AND NOT bPauseSeq AND NOT bQBagHolder THEN bQRBagUp_Down50piston:=TRUE;BagUnitInt:=BagUnitInt+1;END_IF

9:	IF bIBagUpDown50PistonEnd AND NOT bPauseSeq AND NOT bQBagHolder THEN bQRConePusher1Piston:=TRUE;BagUnitInt:=BagUnitInt+1;END_IF

10:	IF bIConePusher1PistonEnd AND NOT bQBagHolder  AND NOT bPauseSeq THEN bQRConePusher1Piston:=FALSE;BagUnitInt:=BagUnitInt+1;END_IF

11:	IF bISeperatorPlatePistonHome  AND NOT bQBagHolder  AND bIConePusher1PistonHome AND NOT bPauseSeq THEN BagUnitInt:=BagUnitInt+1;END_IF

12:	IF  NOT bPauseSeq AND NOT bQBagHolder  THEN BagUnitInt:=BagUnitInt+1;END_IF

13:	BagUnitInt:=BagUnitInt+1;

14:	BagUnitInt:=BagUnitInt+1;

15:	IF bISeperatorPlatePistonHome AND bQRConePusher1Piston AND bIBagUpDown50PistonEnd AND bIBagUpDown180PistonEnd
	AND NOT bQBagHolder  AND NOT bPauseSeq THEN
	bQAColumnStopperPiston:=TRUE;
	bQAConePusher3Piston:= TRUE;
	bQABagUp_Down50piston:=TRUE;
	bQABagUp_Down180piston:=TRUE;
	BagUnitInt:=BagUnitInt+1;
	END_IF

16:	IF bIColumnStopperPistonEnd AND bIBagResetPb  THEN IntAllOver:=TRUE;
	bQRBagUp_Down50piston:=FALSE;
	bQRBagUp_Down180piston:=FALSE;
	BagUnitInt:=0;
	END_IF

END_CASE

IF bMcStopEnable1 OR NOT bAutoModeOn  THEN
bQRBagUp_Down50piston:=FALSE;
bQRBagUp_Down180piston:=FALSE;
bQABagUp_Down50piston:=FALSE;
bQABagUp_Down180piston:=FALSE;
bQAConePusher3Piston:= FALSE;
bQAColumnStopperPiston:=FALSE;
bQRConePusher1Piston:=FALSE;
bQAConePusher1Piston:=FALSE;
bQRBagTiltingpistonForward:=FALSE;
bQRBagTiltingpistonReverse:=FALSE;
bQRBagPusherForwardPiston:= FALSE;
bQRBagPusherReversePiston:=FALSE;
bQRColumnStopperPiston:=FALSE;
bQRColumnReversePiston:=FALSE;
BagUnitInt:=0;
END_IF
END_PROGRAM

(* POU Initialize/ConeFeedCon_Int, ST *)
PROGRAM ConeFeedCon_Int
VAR

	ConeFeedCon: INT;
	bQRConeFeedCon: BOOL;
	bRConePresentInConeFeedCon: BOOL;
	TON_ConeFeedConInt: TON;
	ConeFeedConIntRunning: BOOL;
	sConeFeedConStatus: STRING;
	ConeFeedConIntOver: BOOL;
END_VAR
CASE ConeFeedCon OF

0: IF bAInitializeSeq AND bPauseSeq AND bAutoModeOn THEN
	ConeFeedCon:=ConeFeedCon+1;END_IF

1:	bQRConeFeedCon:=TRUE;ConeFeedCon:=ConeFeedCon+1;

2:	IF bRConePresentInConeFeedCon THEN
		ConeFeedCon:=ConeFeedCon+2;
		ELSIF NOT bRConePresentInConeFeedCon THEN
		ConeFeedCon:=ConeFeedCon+1;
		END_IF

3:	IF  ConeFeedConIntRunning  AND bRConePresentInConeFeedCon THEN
			ConeFeedCon:=ConeFeedCon+1;
	ELSIF TON_ConeFeedConInt.Q  AND NOT bRConePresentInConeFeedCon THEN
		ConeFeedCon:=ConeFeedCon+3;
	END_IF

4:	bQRConeFeedCon:=FALSE;
	TON_ConeFeedConInt(IN:=FALSE);
	ConeFeedCon:=ConeFeedCon+1;

5:	IF NOT bRConePresentInConeFeedCon AND NOT  bPauseSeq THEN
	ConeFeedCon:=1;END_IF

6:	bQRConeFeedCon:=FALSE;
	TON_ConeFeedConInt(IN:=FALSE);
	ConeFeedCon:=ConeFeedCon+1;

7:	ConeFeedConIntOver:=TRUE;
	ConeFeedCon:=ConeFeedCon+1;

8:	ConeFeedCon:=0;

END_CASE

TON_ConeFeedConInt(IN:=bQRConeFeedCon , PT:=T#10s , Q=> , ET=> );

IF TON_ConeFeedConInt.ET >t#1ms AND  TON_ConeFeedConInt.ET<=t#10s THEN
ConeFeedConIntRunning:=TRUE;
ELSE
ConeFeedConIntRunning:=FALSE;
END_IF


IF (bIConeOrientationTopLimitSwitch OR bIUnit_A_ConeCrossLimitSwitch OR bIUnit_B_ConeCrossLimitSwitch)  AND ConeFeedConIntRunning  THEN
bRConePresentInConeFeedCon:=TRUE;
END_IF

IF  bRConePresentInConeFeedCon AND NOT bIConeOrientationTopLimitSwitch AND NOT  bIUnit_A_ConeCrossLimitSwitch
AND NOT  bIUnit_B_ConeCrossLimitSwitch AND bErrorReset THEN bRConePresentInConeFeedCon:=FALSE;END_IF

IF bRConePresentInConeFeedCon THEN
sConeFeedConStatus:='Clear Cone At Cone Feed Conveyor';
ELSE
sConeFeedConStatus:=' Continue Machine Running ';
END_IF

IF bMcStopEnable1 OR NOT bAutoModeOn  THEN
ConeFeedConIntOver:=FALSE;
ConeFeedConIntRunning:=FALSE;
sConeFeedConStatus:=' Continue Machine Running ';
bRConePresentInConeFeedCon:=FALSE;
bQRConeFeedCon:=FALSE;
bAIntHomeCheckError:=FALSE;
IntAllOver:=FALSE;
bAMachineOn:=FALSE;
bAInitializeSeq:=FALSE;
ConeFeedCon:=0;
END_IF
END_PROGRAM

(* POU Initialize/ConeTransfer_Int, ST *)
PROGRAM ConeTransfer_Int
VAR
	ConeTransferInt: INT;

END_VAR
CASE ConeTransferInt OF

0:	IF TiltIntRdy AND NOT bPauseSeq THEN
	ConeTransferInt:=ConeTransferInt+1;END_IF

1:	IF (bITiltingHome OR bITiltingEnd) AND NOT bPauseSeq THEN
	TiltIntRdy:=FALSE;bQRForwardPiston:=TRUE;bQRReversePiston:=TRUE;ConeTransferInt:=ConeTransferInt+1;END_IF

2:	IF bIForwardPistonEnd AND bIReversePistonEnd AND NOT bPauseSeq AND (bITiltingHome OR bITiltingEnd) THEN
	bQRForwardPiston:=FALSE;bQRReversePiston:=FALSE;ConeTransferInt:=ConeTransferInt+1;END_IF

3:	IF bIForwardPistonHome AND bIReversePistonHome AND NOT bPauseSeq THEN
	ConeTransferInt:=ConeTransferInt+1;END_IF

4:	bQRTiltingPiston:=FALSE;
	bQATiltingPiston:=FALSE;
	bQM_Cone_Tilting_Piston:=FALSE;
	bQM_Cone_Tilting_Piston_Rev:=TRUE;
	ConeTransferInt:=ConeTransferInt+1;

5:	IF bITiltingHome AND NOT bPauseSeq THEN
	bQM_Cone_Tilting_Piston_Rev:=FALSE;TiltingIntOvr:=TRUE;ConeTransferInt:=ConeTransferInt+1;END_IF

6:	ConeTransferInt:=0;

END_CASE

IF bMcStopEnable1 OR NOT bAutoModeOn  THEN
TiltingIntOvr:=FALSE;bQRForwardPiston:=FALSE;bQRReversePiston:=FALSE;ConeTransferInt:=0;END_IF
END_PROGRAM

(* POU Initialize/Main_Int, ST *)
PROGRAM Main_Int
VAR
	R_TRIG_1: R_TRIG;
END_VAR
(*************************    INITIAL ERROR CHECK*************************)
IF bMCStartInAuto AND bAutoModeOn   AND NOT bASupplyPressureError
 AND NOT bMcStopEnable AND (bABagModeSelected OR bABoxModeSelected)
	AND NOT IntAllOver  AND NOT bAMainIntStarted THEN  bAMachineOn:=TRUE;END_IF

IF bAInitializeSeq OR bMcStopEnable THEN   bAMachineOn:=FALSE;END_IF

IF bAMachineOn AND NOT bIUnit_A_RowStopperHome THEN bAError1:=TRUE;bAError1Status:='Check Row Stopper A Home';END_IF
IF bAMachineOn AND NOT bIUnit_B_RowStopperHome THEN bAError2:=TRUE;bAError2Status:='Check Row Stopper B Home';END_IF
IF bAMachineOn AND NOT bIConeFeedingPistonHome THEN bAError3:=TRUE;bAError3Status:='Check Cone Feed Piston Home';END_IF
IF bAMachineOn AND NOT bIForwardPistonHome THEN bAError4:=TRUE;bAError4Status:='Check Forward Piston Home';END_IF
IF bAMachineOn AND NOT bIReversePistonHome THEN bAError5:=TRUE;bAError5Status:='Check Reverse Piston  Home';END_IF
IF bAMachineOn AND NOT bITiltingHome THEN bAError6:=TRUE;bAError6Status:='Check Tilting Home';END_IF
IF bAMachineOn AND NOT bIWrappingChanelPiston1Home THEN bAError7:=TRUE;bAError7Status:='Check Wrapping Piston 1  Home';END_IF
IF bAMachineOn AND NOT bIWrappingChanelPiston2Home THEN bAError8:=TRUE;bAError8Status:='Check Wrapping Piston 2 Home';END_IF
IF bAMachineOn AND NOT bISealingTopPistonHome THEN bAError9:=TRUE;bAError9Status:='Check Sealing Top Piston Home';END_IF
IF bAMachineOn AND NOT bISealingBottomPistonHome THEN bAError10:=TRUE;bAError10Status:='Check Sealing Bottom PistonHome';END_IF
IF bAMachineOn AND NOT bISealingSeparatorXAxisPistonHome THEN bAError11:=TRUE;bAError11Status:='Check X Axis Piston Home';END_IF
IF bAMachineOn AND NOT bISealingSeparatorYAxisPistonHome THEN bAError12:=TRUE;bAError12Status:='Check Y Axis Piston Home';END_IF
IF bAMachineOn AND NOT bIColumnStopperPistonHome THEN bAError13:=TRUE;bAError13Status:='Check Column Stopper Home';END_IF
IF bAMachineOn AND NOT bIColumnReversePistonHome THEN bAError14:=TRUE;bAError14Status:='Check Cone Reverse Piston Home';END_IF
IF bAMachineOn AND NOT bISeperatorPlatePistonHome THEN bAError15:=TRUE;bAError15Status:='Check Seperator Piston Home';END_IF
IF bAMachineOn AND NOT bIConePusher1PistonHome THEN bAError16:=TRUE;bAError16Status:='Check Cone Pusher 2 Home';END_IF
IF bAMachineOn AND NOT bIBagUpDown50PistonHome THEN bAError17:=TRUE;bAError17Status:='Check Up Down Piston 50 Home';END_IF
IF bAMachineOn AND NOT bIBagUpDown180PistonHome THEN bAError18:=TRUE;bAError18Status:='Check Up Down Piston 180 Home';END_IF
IF bAMachineOn AND NOT bIBagPusherPistonHome THEN bAError19:=TRUE;bAError19Status:='Check Bag Pusher Home';END_IF
IF bAMachineOn AND NOT bIBagTiltingPistonHome THEN bAError20:=TRUE;bAError20Status:='Check Bag Tilting Home';END_IF

IF bErrorReset AND bAMachineOn AND bIUnit_A_RowStopperHome  AND NOT IntAllOver THEN bAError1:=FALSE;bAError1Status:='Continue Machine Running';END_IF

IF bErrorReset AND bAMachineOn AND bIUnit_B_RowStopperHome  AND NOT IntAllOver THEN bAError2:=FALSE;bAError2Status:='Continue Machine Running';END_IF

IF bErrorReset AND bAMachineOn AND bIConeFeedingPistonHome  AND NOT IntAllOver THEN bAError3:=FALSE;bAError3Status:='Continue Machine Running';END_IF

IF bErrorReset AND bAMachineOn AND bIForwardPistonHome  AND NOT IntAllOver THEN bAError4:=FALSE;bAError4Status:='Continue Machine Running';END_IF

IF bErrorReset AND bAMachineOn AND bIReversePistonHome  AND NOT IntAllOver THEN bAError5:=FALSE;bAError5Status:='Continue Machine Running';END_IF

IF bErrorReset AND bAMachineOn AND bITiltingHome  AND NOT IntAllOver THEN bAError6:=FALSE;bAError6Status:='Continue Machine Running';END_IF

IF bErrorReset AND bAMachineOn AND bIWrappingChanelPiston1Home  AND NOT IntAllOver THEN bAError7:=FALSE;bAError7Status:='Continue Machine Running';END_IF

IF bErrorReset AND bAMachineOn AND bIWrappingChanelPiston2Home  AND NOT IntAllOver THEN bAError8:=FALSE;bAError8Status:='Continue Machine Running';END_IF

IF bErrorReset AND bAMachineOn AND bISealingTopPistonHome  AND NOT IntAllOver THEN bAError9:=FALSE;bAError9Status:='Continue Machine Running';END_IF

IF bErrorReset AND bAMachineOn AND bISealingBottomPistonHome  AND NOT IntAllOver THEN bAError10:=FALSE;bAError10Status:='Continue Machine Running';END_IF

IF bErrorReset AND bAMachineOn AND bISealingSeparatorXAxisPistonHome  AND NOT IntAllOver THEN bAError11:=FALSE;bAError11Status:='Continue Machine Running';END_IF

IF bErrorReset AND bAMachineOn AND bISealingSeparatorYAxisPistonHome   AND NOT IntAllOver THEN bAError12:=FALSE;bAError12Status:='Continue Machine Running';END_IF

IF bErrorReset AND bAMachineOn AND bIColumnStopperPistonHome  AND NOT IntAllOver THEN bAError13:=FALSE;bAError13Status:='Continue Machine Running';END_IF

IF bErrorReset AND bAMachineOn AND bIColumnReversePistonHome  AND NOT IntAllOver THEN bAError14:=FALSE;bAError14Status:='Continue Machine Running';END_IF

IF bErrorReset AND bAMachineOn AND bISeperatorPlatePistonHome  AND NOT IntAllOver THEN bAError15:=FALSE;bAError15Status:='Continue Machine Running';END_IF

IF bErrorReset AND bAMachineOn AND bIConePusher1PistonHome  AND NOT IntAllOver THEN bAError16:=FALSE;bAError16Status:='Continue Machine Running';END_IF

IF bErrorReset AND bAMachineOn AND bIBagUpDown50PistonHome  AND NOT IntAllOver THEN bAError17:=FALSE;bAError17Status:='Continue Machine Running';END_IF

IF bErrorReset AND bAMachineOn AND bIBagUpDown180PistonHome  AND NOT IntAllOver THEN bAError18:=FALSE;bAError18Status:='Continue Machine Running';END_IF

IF bErrorReset AND bAMachineOn AND bIBagPusherPistonHome  AND NOT IntAllOver THEN bAError19:=FALSE;bAError19Status:='Continue Machine Running';END_IF

IF bErrorReset AND bAMachineOn AND bIBagTiltingPistonHome  AND NOT IntAllOver THEN bAError20:=FALSE;bAError20Status:='Continue Machine Running';END_IF


										(***MAIN INT***)
IF Initialize_TapHmi  AND bMcStartInAuto AND bAutoModeOn AND NOT bASupplyPressureError
	 AND (bABagModeSelected OR bABoxModeSelected) AND NOT bAIntHomeCheckError
	AND NOT IntAllOver AND NOT  bMcStopEnable AND NOT bAMainIntStarted THEN
	bAInitializeSeq:=TRUE;
	bAMainIntStarted:=TRUE;
ELSE
	bAInitializeSeq:=FALSE;
END_IF


	R_TRIG_1(CLK:= IntAllOver  , Q=> );
IF  bMcStopEnable OR R_TRIG_1.Q   OR NOT bAutoModeOn  THEN bAMainIntStarted:=FALSE; END_IF
END_PROGRAM

(* POU Initialize/Ret_Int, ST *)
PROGRAM Ret_Int
VAR
	Ret_A_Int: INT;
	bQRRetA_RowStopperMotorRev: BOOL;
	Ret_B_Int: INT;
	bQRRetB_RowStopperMotorRev: BOOL;
END_VAR
					(*********************Ret-A Int Logic****************)
CASE Ret_A_Int OF

0:IF bIMcStartPb AND NOT bAMainIntStarted THEN
	Ret_A_Int:=Ret_A_Int+1;END_IF

1:IF bIUnit_A_RowStopperHome THEN Ret_A_Int:=Ret_A_Int+2;
	ELSIF NOT bIUnit_A_RowStopperHome THEN Ret_A_Int:=Ret_A_Int+1;END_IF

2:bQRRetA_RowStopperMotorRev:=TRUE;Ret_A_Int:=Ret_A_Int+1;

3:IF bIUnit_A_RowStopperHome THEN
	bQRRetA_RowStopperMotorRev:=FALSE;Ret_A_Int:=Ret_A_Int+1;END_IF

4:Ret_A_Int:=0;

END_CASE


					(*********************Ret-B Int Logic****************)
CASE Ret_B_Int OF

0:IF bIMcStartPb AND NOT bAMainIntStarted THEN
	Ret_B_Int:=Ret_B_Int+1;END_IF

1:IF bIUnit_B_RowStopperHome THEN Ret_B_Int:=Ret_B_Int+2;
	ELSIF NOT bIUnit_B_RowStopperHome THEN Ret_B_Int:=Ret_B_Int+1;END_IF

2:bQRRetB_RowStopperMotorRev:=TRUE;Ret_B_Int:=Ret_B_Int+1;

3:IF bIUnit_B_RowStopperHome THEN
	bQRRetB_RowStopperMotorRev:=FALSE;Ret_B_Int:=Ret_B_Int+1;END_IF

4:Ret_B_Int:=0;

END_CASE
END_PROGRAM

(* POU Initialize/Sealing_Int, ST *)
PROGRAM Sealing_Int
VAR
	SealConInt:INT;
	TON_SealingConInt:TON;
	SealingPistonInt:INT;
	BagIntCheck:INT;
	TON_SealingPis:TON;
	TON_SealingDly_Int:TON;


END_VAR
CASE SealConInt OF

0:IF WrapUnitIntOver AND NOT bPauseSeq AND bAutoModeOn THEN
	SealConInt:=SealConInt+1;END_IF

1:IF WrappingSafety AND NOT bPauseSeq THEN
	bQRSealingConveyorMotor:=TRUE;WrapUnitIntOver:=FALSE;SealConInt:=SealConInt+1;END_IF

2:	IF bRConePresentInSealCon THEN
		SealConInt:=SealConInt+2;
		ELSIF NOT bRConePresentInSealCon THEN
		SealConInt:=SealConInt+1;
		END_IF

3:IF  SealingConIntRunning  AND bRConePresentInSealCon THEN
			SealConInt:=SealConInt+1;
	ELSIF TON_SealingConInt.Q  AND NOT bRConePresentInSealCon THEN
		SealConInt:=SealConInt+3;
	END_IF

4:	bQRSealingConveyorMotor:=FALSE;
	TON_SealingConInt(IN:=FALSE);
	SealConInt:=SealConInt+1;

5:	IF NOT bRConePresentInSealCon AND NOT  bPauseSeq THEN
	SealConInt:=1;END_IF

6:	bQRSealingConveyorMotor:=FALSE;
	TON_SealingConInt(IN:=FALSE);
	SealConInt:=SealConInt+1;

7:	SealConIntOver:=TRUE;
	SealConInt:=SealConInt+1;

8:	SealConInt:=0;

END_CASE


TON_SealingConInt(IN:=bQRSealingConveyorMotor , PT:=T#10s , Q=> , ET=> );

IF TON_SealingConInt.ET >t#1ms AND  TON_SealingConInt.ET<=t#10s THEN
SealingConIntRunning:=TRUE;
ELSE
SealingConIntRunning:=FALSE;
END_IF


IF bIConeCountsensor  AND SealingConIntRunning  THEN
bRConePresentInSealCon:=TRUE;
END_IF

IF  bRConePresentInSealCon AND NOT bIConeCountsensor
AND bErrorReset THEN bRConePresentInSealCon:=FALSE;END_IF

IF bRConePresentInSealCon THEN
sSealingConStatus:='Clear Cone At Sealing Conveyor';
ELSE
sSealingConStatus:=' Continue Machine Running ';
END_IF

CASE SealingPistonInt OF

0:	IF SealConIntOver AND WrappingSafety AND NOT bPauseSeq AND bAutoModeOn THEN
	bQRSealingSeparatorYAxisPiston:=TRUE;SealingPistonInt:=SealingPistonInt+1;END_IF

1:	IF bISealingSeparatorYAxisPistoEnd AND NOT bPauseSeq THEN
	bQRSealingTopPiston:=TRUE;bQRSealingBottomPiston:=TRUE;SealingPistonInt:=SealingPistonInt+1;END_IF

2:	TON_SealingPis(IN:=TRUE , PT:=t#2s , Q=> , ET=> );
	IF (bISealingTopPistonEnd AND bISealingBottomPistonEnd) OR TON_SealingPis.Q THEN
	SealingPistonInt:=SealingPistonInt+1;END_IF

3:	TON_SealingDly_Int(IN:=TRUE , PT:= t#2s, Q=> , ET=> );
	IF TON_SealingDly_Int.Q THEN SealingPistonInt:=SealingPistonInt+1;END_IF

4:	bQRSealingSeparatorXAxisPiston:=TRUE;TON_SealingPis(IN:=FALSE);TON_SealingDly_Int(IN:=FALSE);
	SealingPistonInt:=SealingPistonInt+1;

5:	IF bISealingSeparatorXAxisPistonEnd AND NOT bPauseSeq THEN
	bQRSealingSeparatorYAxisPiston:=FALSE;
	bQRSealingTopPiston:=FALSE;bQRSealingBottomPiston:=FALSE;
	bQRSealingSeparatorXAxisPiston:=FALSE;SealingPistonInt:=SealingPistonInt+1;END_IF

6:	IF SealingSafety AND NOT bPauseSeq THEN
	bRSealUnitIntOver:=TRUE;SealingPistonInt:=SealingPistonInt+1;END_IF

7:	SealingPistonInt:=0;

END_CASE

CASE BagIntCheck OF

0: 	IF bABagModeSelected AND NOT bPauseSeq AND bRSealUnitIntOver AND TiltingIntOvr THEN
	bRBagUnitIntRdy:=TRUE;
	ELSIF bABoxModeSelected AND NOT bPauseSeq AND bRSealUnitIntOver AND TiltingIntOvr THEN
	IntAllOver:=TRUE;bRSealUnitIntOver:=FALSE; TiltingIntOvr:=FALSE;BagIntCheck:=BagIntCheck+1;END_IF

1:	BagIntCheck:=0;
END_CASE;


IF bMcStopEnable1 OR NOT bAutoModeOn  THEN
bRSealUnitIntOver:=FALSE;SealingPistonInt:=0;bQRSealingSeparatorYAxisPiston:=FALSE;
	bQRSealingTopPiston:=FALSE;bQRSealingBottomPiston:=FALSE;
	bQRSealingSeparatorXAxisPiston:=FALSE;TON_SealingDly_Int(IN:=FALSE);
TON_SealingPis(IN:=FALSE);SealConIntOver:=FALSE;SealingConIntRunning:=FALSE;
bRConePresentInSealCon:=FALSE;TON_SealingConInt(IN:=FALSE);
bQRSealingConveyorMotor:=FALSE;WrapUnitIntOver:=FALSE;SealConInt:=0;BagIntCheck:=0;
END_IF
END_PROGRAM

(* POU Initialize/Wrapping_Int, ST *)
PROGRAM Wrapping_Int
VAR
	WrapConInt: INT;

	TON_WrappingConInt: TON;
	WrapPistonInt: INT;


END_VAR
CASE WrapConInt OF

0:IF bAInitializeSeq AND NOT bPauseSeq AND bAutoModeOn THEN
	WrapConInt:=WrapConInt+1;END_IF

1:IF WrappingSafety AND NOT bPauseSeq THEN
	bQRWappingConveyorMotor:=TRUE;WrapConInt:=WrapConInt+1;END_IF

2:	IF bRConePresentInWrapCon THEN
		WrapConInt:=WrapConInt+2;
		ELSIF NOT bRConePresentInWrapCon THEN
		WrapConInt:=WrapConInt+1;
		END_IF

3:IF  WrappingConIntRunning  AND bRConePresentInWrapCon THEN
			WrapConInt:=WrapConInt+1;
	ELSIF TON_WrappingConInt.Q  AND NOT bRConePresentInWrapCon THEN
		WrapConInt:=WrapConInt+3;
	END_IF

4:	bQRWappingConveyorMotor:=FALSE;
	TON_WrappingConInt(IN:=FALSE);
	WrapConInt:=WrapConInt+1;

5:	IF NOT bRConePresentInWrapCon AND NOT  bPauseSeq THEN
	WrapConInt:=1;END_IF

6:	bQRWappingConveyorMotor:=FALSE;
	TON_WrappingConInt(IN:=FALSE);
	WrapConInt:=WrapConInt+1;

7:	WrapConIntOver:=TRUE;
	TiltIntRdy:=TRUE;
	WrapConInt:=WrapConInt+1;

8:	WrapConInt:=0;

END_CASE


TON_WrappingConInt(IN:=bQRWappingConveyorMotor , PT:=T#10s , Q=> , ET=> );

IF TON_WrappingConInt.ET >t#1ms AND  TON_WrappingConInt.ET<=t#10s THEN
WrappingConIntRunning:=TRUE;
ELSE
WrappingConIntRunning:=FALSE;
END_IF


IF (bIWrappingCone1 OR bIWrappingCone1)  AND WrappingConIntRunning  THEN
bRConePresentInWrapCon:=TRUE;
END_IF

IF  bRConePresentInWrapCon AND NOT bIWrappingCone1 AND NOT  bIWrappingCone2
AND bErrorReset THEN bRConePresentInWrapCon:=FALSE;END_IF

IF bRConePresentInWrapCon THEN
sWrappingConStatus:='Clear Cone At Wrapping Conveyor';
END_IF

CASE WrapPistonInt OF

0:	IF WrapConIntOver AND NOT bPauseSeq AND SealingSafety THEN
	bQRWrappingPiston1:=TRUE;bQRWrappingPiston2:=TRUE;WrapConIntOver:=FALSE;WrapPistonInt:=WrapPistonInt+1;END_IF

1:	 IF NOT bPauseSeq AND NOT bAWrappingPiston1RsError AND NOT bAWrappingPiston2RsError AND
	bIWrappingChanelPiston1End AND bIWrappingChanelPiston2End THEN
	bQRWrappingPiston1:=FALSE;bQRWrappingPiston2:=FALSE;WrapPistonInt:=WrapPistonInt+1;END_IF

2:	 IF  NOT bPauseSeq AND WrappingSafety THEN
	WrapUnitIntOver:=TRUE;WrapPistonInt:=WrapPistonInt+1;END_IF

3:	WrapPistonInt:=0;

END_CASE


IF bMcStopEnable1 OR NOT bAutoModeOn  THEN
WrapPistonInt:=0;WrapConIntOver:=FALSE;bAWrappingPiston1RsError:=FALSE;bAWrappingPiston2RsError:=FALSE;
bQRWrappingPiston1:=FALSE;bQRWrappingPiston2:=FALSE;WrapUnitIntOver:=FALSE;
WrappingConIntRunning:=FALSE;bRConePresentInWrapCon:=FALSE;WrapConInt:=0;TON_WrappingConInt(IN:=FALSE);
bQRWappingConveyorMotor:=FALSE;END_IF
END_PROGRAM

(* POU Manual, ST *)
PROGRAM Manual
VAR

	step: INT;
	Timer1: TON;

END_VAR
					(*************SEALING SAFETY*********************)

IF	bISealingTopPistonHome AND bISealingBottomPistonHome AND bISealingSeparatorYAxisPistonHome AND bISealingSeparatorXAxisPistonHome
THEN
	SealingSafety:=TRUE;
ELSE
	SealingSafety:=FALSE;
END_IF

						(*************WRAPPING  SAFETY*********************)
IF 	bIWrappingChanelPiston1Home AND  bIWrappingChanelPiston2Home
THEN
	WrappingSafety:=TRUE;
ELSE
	WrappingSafety:=FALSE;
END_IF

					(*======================MANUAL SEALING LOGIC==========================*)

IF NOT  bAutoModeOn AND bIManualSealingPb THEN
	bManualSealEnable:=TRUE;
ELSE bManualSealEnable:=FALSE; END_IF

IF   bAutoModeOn AND bPauseSeq  AND bIManualSealingPb THEN
bManualSealEnable2:=TRUE;
ELSE bManualSealEnable2:=FALSE; END_IF

CASE step OF

	0:	IF  ( bManualSealEnable OR bManualSealEnable2  )THEN bMManualSealOn:=TRUE; step:=step+1;  END_IF

	1:	Timer1(IN:= FALSE);
		bQM_Cone_Sealing_Bottom_Piston:=TRUE;
		bQM_Cone_Sealing_Top_Piston:=TRUE;
		step:=step+1;

	2:	 IF bISealingBottomPistonEnd AND bISealingTopPistonEnd THEN
		 step:=step+1;
		END_IF

	3:	Timer1(IN:=TRUE , PT:=t#3s , Q=> , ET=> );
		IF Timer1.Q THEN step:=step+1; END_IF

	4:	bMManualSealOn:=FALSE;
		bQM_Cone_Sealing_Bottom_Piston:=FALSE;
		bQM_Cone_Sealing_Top_Piston:=FALSE;
		Timer1(IN:= FALSE);
		 step:=step+1;

	5:	step:=0;
END_CASE

								(*************RET-A FWD ; REV *********************)
IF bHMI_RetA_Fwd_On AND NOT bHMI_RetA_Rev_On AND NOT  bQM_RetA_Rev THEN bQM_RetA_Fwd:=TRUE;ELSE bQM_RetA_Fwd:=FALSE;END_IF

IF bHMI_Ret_RevA_On AND NOT bHMI_RetA_Fwd_On AND NOT bQM_RetA_Fwd THEN bQM_RetA_Rev:=TRUE;ELSE bQM_RetA_Rev:=FALSE;END_IF



								(*************RET-A FWD ; REV *********************)
IF bHMI_RetB_Fwd_On AND NOT bHMI_RetB_Rev_On AND NOT  bQM_RetB_Rev THEN bQM_RetB_Fwd:=TRUE;ELSE bQM_RetB_Fwd:=FALSE;END_IF

IF bHMI_Ret_RevB_On AND NOT bHMI_RetB_Fwd_On AND NOT bQM_RetB_Fwd THEN bQM_RetB_Rev:=TRUE;ELSE bQM_RetB_Rev:=FALSE;END_IF



								(*************CONE FEEDING PISTON*********************)
IF bHMI_Cone_Feeding_Piston_On THEN
	bQM_Cone_Feeding_Piston:=TRUE;
ELSE bQM_Cone_Feeding_Piston:=FALSE;END_IF

								(*************CONE FORWARD PISTON*********************)
IF bHMI_Cone_Forward_Piston_On THEN
bQM_Cone_Forward_Piston:=TRUE;
ELSE bQM_Cone_Forward_Piston:=FALSE;END_IF

								(*************CONE REVERSE PISTON*********************)
IF bHMI_Cone_Reverse_Piston_On THEN
bQM_Cone_Reverse_Piston:=TRUE;
ELSE bQM_Cone_Reverse_Piston:=FALSE;END_IF

								(*************CONE TILTING PISTON*********************)
IF bHMI_Cone_Tilting_Piston_On THEN
bQM_Cone_Tilting_Piston:=TRUE;bQM_Cone_Tilting_Piston_Rev:=FALSE;
ELSE bQM_Cone_Tilting_Piston:=FALSE;END_IF
IF bHMI_Cone_Tilting_Piston_On_Rev THEN
bQM_Cone_Tilting_Piston:=FALSE;bQM_Cone_Tilting_Piston_Rev:=TRUE;
ELSE bQM_Cone_Tilting_Piston_Rev:=FALSE;END_IF

								(*************WRAPPING PISTON 1*********************)
IF bHMI_Cone_Wrapping_Piston1_On AND SealingSafety THEN
bQM_Cone_Wrapping_Piston1_Rev:=FALSE;bQM_Cone_Wrapping_Piston1_Fwd:=TRUE;
ELSE bQM_Cone_Wrapping_Piston1_Fwd:=FALSE;END_IF

IF bHMI_Cone_Wrapping_Piston1_On_Rev AND SealingSafety THEN
bQM_Cone_Wrapping_Piston1_Fwd:=FALSE;bQM_Cone_Wrapping_Piston1_Rev:=TRUE;
ELSE bQM_Cone_Wrapping_Piston1_Rev:=FALSE;END_IF

					(*************WRAPPING PISTON 2*********************)
IF bHMI_Cone_Wrapping_Piston2_On AND SealingSafety THEN
bQM_Cone_Wrapping_Piston2_Rev:=FALSE;bQM_Cone_Wrapping_Piston2_Fwd:=TRUE;
ELSE bQM_Cone_Wrapping_Piston2_Fwd:=FALSE;END_IF

IF bHMI_Cone_Wrapping_Piston2_On_Rev AND SealingSafety THEN
bQM_Cone_Wrapping_Piston2_Fwd:=FALSE;bQM_Cone_Wrapping_Piston2_Rev:=TRUE;
ELSE bQM_Cone_Wrapping_Piston2_Rev:=FALSE;END_IF


								(*************SEALING TOP PISTON*********************)
IF bHMI_Cone_Sealing_Top_Piston_On AND WrappingSafety THEN
bQM_Cone_Sealing_Top_Piston:=TRUE;ELSE bQM_Cone_Sealing_Top_Piston:=FALSE;END_IF


								(*************SEALING BOTTOM PISTON*********************)
IF bHMI_Cone_Sealing_Bottom_Piston_On AND WrappingSafety THEN
bQM_Cone_Sealing_Bottom_Piston:=TRUE;
ELSE bQM_Cone_Sealing_Bottom_Piston:=FALSE;END_IF


								(*************SEALING Y AXIS  PISTON*********************)
IF bHMI_Cone_Sealing_YAxis_Piston_On AND WrappingSafety THEN
bQM_Cone_Sealing_YAxis_Piston:=TRUE;ELSE bQM_Cone_Sealing_YAxis_Piston:=FALSE;END_IF


								(*************SEALING X AXIS  PISTON*********************)
IF bHMI_Cone_Sealing_XAxis_Piston_On AND WrappingSafety THEN
bQM_Cone_Sealing_XAxis_Piston:=TRUE;ELSE bQM_Cone_Sealing_XAxis_Piston:=FALSE;END_IF

								(*************CONE FEEDING CONVEYOR MOTOR*********************)
IF bHMI_Cone_Feeding_Conveyor_On THEN
bQM_Cone_Feeding_Conveyor:=TRUE;
ELSE bQM_Cone_Feeding_Conveyor:=FALSE;END_IF


								(*************CONE WRAPPING CONVEYOR MOTOR*********************)
IF bHMI_Cone_Wrapping_Conveyor_On THEN
bQM_Cone_Wrapping_Conveyor:=TRUE;ELSE bQM_Cone_Wrapping_Conveyor:=FALSE;END_IF


								(*************CONE SEALING CONVEYOR MOTOR*********************)
IF bHMI_Cone_Sealing_Conveyor_On THEN
bQM_Cone_Sealing_Conveyor:=TRUE;
ELSE bQM_Cone_Sealing_Conveyor:=FALSE;END_IF



										(***CONE PUSHER 1***)
IF bIConePusher1_On_Hmi THEN
bQMConePusher1:=TRUE;
ELSE bQMConePusher1:=FALSE;END_IF


										(***CONE PUSHER 2***)
IF bIConePusher2_On_Hmi THEN
bQMConePusher2:=TRUE;ELSE
bQMConePusher2:=FALSE;END_IF


										(***CONE PUSHER 3***)
IF bIConePusher3_On_Hmi THEN
bQMConePusher3:=TRUE;
ELSE bQMConePusher3:=FALSE;END_IF


										(***BAG PUSHER FORWARD***)
IF bIBagPusherFwd_On_Hmi THEN
bQMBagPusherFwd:=TRUE;
ELSE bQMBagPusherFwd:=FALSE;END_IF


										(***BAG PUSHER REVERSE***)
IF bIBagPusherRev_On_Hmi THEN
bQMBagPusherRev:=TRUE;
ELSE bQMBagPusherRev:=FALSE;END_IF


										(***UP DOWN PISTON 1***)
IF bIUpDownPiston_1_On_Hmi THEN
bQMUpDownPiston_1:=TRUE;
ELSE bQMUpDownPiston_1:=FALSE;END_IF


										(***UP DOWN PISTON 2***)
IF bIUpDownPiston_2_On_Hmi THEN
bQMUpDownPiston_2:=TRUE;
ELSE bQMUpDownPiston_2:=FALSE;END_IF



										(***BAG TILTING FORWARD***)
IF bIBagTiltingFwd_On_Hmi THEN
bQMBagTiltingFwd:=TRUE;
ELSE bQMBagTiltingFwd:=FALSE;END_IF


										(***BAG TILTING REVERSE***)
IF bIBagTiltingRev_On_Hmi THEN
bQMBagTiltingRev:=TRUE;
ELSE bQMBagTiltingRev:=FALSE;END_IF


										(***bQRColumn Stopper Piston ***)
IF bIColumn_Stopper_Piston_On_Hmi THEN
bQMColumnStopperPiston:=TRUE;
ELSE bQMColumnStopperPiston:=FALSE;END_IF


										(***bQRColumn Stopper Piston ***)
IF bIColumnConeForwardPiston_On_Hmi THEN
bQMColumnConeForwardPiston:=TRUE;
ELSE bQMColumnConeForwardPiston:=FALSE;END_IF


																(***BAG HOLDER ***)
IF   (bAutoModeOn    AND (bIBagHolder_On OR bIBagHolder_On_Hmi)
AND bIBagPusherHome) OR (bManualModeOn AND  (bIBagHolder_On OR bIBagHolder_On_Hmi) AND bIBagPusherHome) THEN
bQMBagHolderPiston:=TRUE;
ELSE bQMBagHolderPiston:=FALSE;END_IF



IF bMcStopEnable1 OR NOT bManualModeOn  THEN
	bHMI_RetA_Fwd_On:=FALSE;
	bHMI_RetA_Rev_On:=FALSE;
	bHMI_RetB_Fwd_On:=FALSE;
	bHMI_RetB_Rev_On:=FALSE;
	bHMI_Cone_Feeding_Piston_On  :=FALSE;
	bHMI_Cone_Forward_Piston_On:=FALSE;
	bHMI_Cone_Reverse_Piston_On :=FALSE;
	bHMI_Cone_Tilting_Piston_On :=FALSE;
	bHMI_Cone_Wrapping_Piston1_On :=FALSE;
	bHMI_Cone_Wrapping_Piston2_On :=FALSE;
	bHMI_Cone_Sealing_YAxis_Piston_On :=FALSE;
	bHMI_Cone_Sealing_XAxis_Piston_On :=FALSE;
	bHMI_Cone_Sealing_Top_Piston_On :=FALSE;
	bHMI_Cone_Sealing_Bottom_Piston_On :=FALSE;
	bHMI_Cone_Feeding_Conveyor_On :=FALSE;
	bHMI_Cone_Wrapping_Conveyor_On :=FALSE;
	bHMI_Cone_Sealing_Conveyor_On :=FALSE;
	bQM_RetB_Fwd:=FALSE;
	bQM_RetB_Rev:=FALSE;
	bQM_Cone_Feeding_Piston:=FALSE;
	bQM_Cone_Forward_Piston:=FALSE;
	bQM_Cone_Reverse_Piston:=FALSE;
	bQM_Cone_Sealing_YAxis_Piston:=FALSE;
	bQM_Cone_Sealing_XAxis_Piston:=FALSE;
	bQM_Cone_Feeding_Conveyor:=FALSE;
 	bQM_Cone_Wrapping_Conveyor:=FALSE;
	bQM_Cone_Sealing_Conveyor:=FALSE;
	bQMConePusher1:=FALSE;
	bQMConePusher2:=FALSE;
	bQMConePusher3:=FALSE;
	bQMBagPusherFwd:=FALSE;
	bQMBagPusherRev:=FALSE;
	bQMUpDownPiston_1:=FALSE;
	bQMUpDownPiston_2:=FALSE;
	bQMBagTiltingFwd:=FALSE;
	bQMBagTiltingRev:=FALSE;
	bQMColumnStopperPiston:=FALSE;
	bQMColumnConeForwardPiston:=FALSE;
	bQM_RetA_Rev:=FALSE;
	bQM_RetA_Fwd:=FALSE;
	bQM_RetB_Rev:=FALSE;
	bQM_RetB_Fwd:=FALSE;
	bIConePusher1_On_Hmi:=FALSE;
	bIConePusher2_On_Hmi:=FALSE;
	bIConePusher3_On_Hmi:=FALSE;
	bIBagPusherFwd_On_Hmi:=FALSE;
	bIBagPusherRev_On_Hmi:=FALSE;
	bIUpDownPiston_1_On_Hmi:=FALSE;
	bIUpDownPiston_2_On_Hmi:=FALSE;
	bIBagTiltingFwd_On_Hmi:=FALSE;
	bIBagTiltingRev_On_Hmi:=FALSE;
	bIColumn_Stopper_Piston_On_Hmi:=FALSE;
	bIColumnConeForwardPiston_On_Hmi:=FALSE;
	bIBagHolder_On_Hmi:=FALSE;
	bQM_Cone_Sealing_Top_Piston:=FALSE;
	bQM_Cone_Sealing_Bottom_Piston:=FALSE;
	step:=0;
END_IF
END_PROGRAM

(* POU Weight_Read, ST *)
PROGRAM Weight_Read
VAR
	COMportControl_1: SerialLineControl;
	COMin_1_COMPort_1 AT %I*: EL6inData22B;
	COMOut_1_COMPort_1 AT %Q*: EL6outData22B;
	TxBuffer1: ComBuffer;
	RxBuffer1: ComBuffer;
	ipos_1: INT;
	samplestring_1: STRING;
	ReceiveString_sample_1: ReceiveString;
	resultWt_1: STRING;
	COMportControlError_1: BOOL;
	COMportControlErrorID_1: ComError_t;
	Ret_AWt: REAL;


	COMportControl_2: SerialLineControl;
	COMin_2_COMPort_2 AT %I*: EL6inData22B;
	COMOut_2_COMPort_2 AT %Q*: EL6outData22B;
	TxBuffer2: ComBuffer;
	RxBuffer2: ComBuffer;
	ipos_2: INT;
	samplestring_2: STRING;
	ReceiveString_sample_2: ReceiveString;
	resultWt_2: STRING;
	COMportControlError_2: BOOL;
	COMportControlErrorID_2: ComError_t;
	Ret_BWt: REAL;

END_VAR
(*==============Ret - A Weight Read==================*)

COMportControl_1(
	Mode:= SERIALLINEMODE_EL6_22B,
	pComIn:= ADR(COMin_1_COMport_1),
	pComOut:= ADR(COMout_1_COMport_1),
	SizeComIn:= SIZEOF(COMin_1_COMport_1),
	TxBuffer:= TxBuffer1,
	RxBuffer:= RxBuffer1,
	Error=> COMportControlError_1,
	ErrorID=> COMportControlErrorID_1);

